  MoveL 1972 to (51.44, -54.38, -208.01) mm, rotated rx -9.61 ry -16.54 rz 125.97 deg; joints [-13.21, -58.037, 110.38, 194.099, 36.852, -114.104, -235]
  MoveL 1973 to (50.7, -54.44, -208.96) mm, rotated rx -9.61 ry -16.54 rz 125.97 deg; joints [-13.251, -58.035, 110.423, 194.018, 36.888, -114.045, -235]
  MoveL 1974 to (50.05, -54.2, -209.74) mm, rotated rx -9.61 ry -16.54 rz 125.97 deg; joints [-13.287, -58.053, 110.472, 193.952, 36.914, -113.997, -235]
  MoveL 1975 to (49.76, -53.97, -210.06) mm, rotated rx -9.61 ry -16.54 rz 125.97 deg; joints [-13.302, -58.07, 110.5, 193.925, 36.922, -113.978, -235]
  MoveL 1976 to (49.49, -53.67, -210.35) mm, rotated rx -9.61 ry -16.54 rz 125.97 deg; joints [-13.316, -58.091, 110.529, 193.901, 36.928, -113.961, -235]
  MoveL 1977 to (49.02, -52.84, -210.78) mm, rotated rx -9.61 ry -16.54 rz 125.97 deg; joints [-13.338, -58.15, 110.594, 193.863, 36.931, -113.936, -235]
  MoveL 1978 to (48.65, -51.71, -211.04) mm, rotated rx -9.61 ry -16.54 rz 125.97 deg; joints [-13.354, -58.228, 110.666, 193.839, 36.922, -113.923, -235]
  MoveL 1979 to (48.37, -50.29, -211.12) mm, rotated rx -9.61 ry -16.54 rz 125.97 deg; joints [-13.364, -58.326, 110.745, 193.83, 36.902, -113.921, -235]
  MoveL 1980 to (48.3, -49.77, -211.12) mm, rotated rx -9.61 ry -16.54 rz 125.97 deg; joints [-13.366, -58.362, 110.773, 193.829, 36.894, -113.922, -235]
  MoveL 1981 to (48.25, -49.32, -211.1) mm, rotated rx -9.61 ry -16.54 rz 125.97 deg; joints [-13.367, -58.393, 110.795, 193.831, 36.885, -113.925, -235]
  MoveL 1982 to (48.22, -48.89, -211.05) mm, rotated rx -9.61 ry -16.54 rz 125.97 deg; joints [-13.367, -58.422, 110.816, 193.834, 36.877, -113.928, -235]
  MoveL 1983 to (48.2, -48.47, -210.99) mm, rotated rx -9.61 ry -16.54 rz 125.97 deg; joints [-13.366, -58.451, 110.835, 193.838, 36.868, -113.933, -235]
  MoveL 1984 to (48.17, -48.02, -210.95) mm, rotated rx -9.61 ry -16.54 rz 125.97 deg; joints [-13.366, -58.482, 110.857, 193.841, 36.859, -113.936, -235]
  MoveL 1985 to (48.11, -47.51, -210.94) mm, rotated rx -9.61 ry -16.54 rz 125.97 deg; joints [-13.367, -58.517, 110.883, 193.842, 36.85, -113.939, -235]
  MoveL 1986 to (48.03, -47, -210.94) mm, rotated rx -9.61 ry -16.54 rz 125.97 deg; joints [-13.37, -58.553, 110.91, 193.841, 36.841, -113.94, -235]
  MoveL 1987 to (47.96, -46.5, -210.93) mm, rotated rx -9.61 ry -16.54 rz 125.97 deg; joints [-13.371, -58.587, 110.936, 193.841, 36.833, -113.941, -235]
  MoveL 1988 to (47.9, -46.03, -210.91) mm, rotated rx -9.61 ry -16.54 rz 125.97 deg; joints [-13.372, -58.619, 110.96, 193.842, 36.825, -113.944, -235]
  MoveL 1989 to (47.87, -45.61, -210.85) mm, rotated rx -9.61 ry -16.54 rz 125.97 deg; joints [-13.372, -58.649, 110.981, 193.845, 36.817, -113.948, -235]
  MoveL 1990 to (47.84, -45.19, -210.79) mm, rotated rx -9.61 ry -16.54 rz 125.97 deg; joints [-13.371, -58.678, 111.001, 193.849, 36.808, -113.952, -235]
  MoveL 1991 to (47.81, -44.72, -210.74) mm, rotated rx -9.61 ry -16.54 rz 125.97 deg; joints [-13.371, -58.71, 111.024, 193.853, 36.799, -113.956, -235]
  MoveL 1992 to (47.74, -44.11, -210.7) mm, rotated rx -9.61 ry -16.54 rz 125.97 deg; joints [-13.372, -58.752, 111.054, 193.855, 36.787, -113.96, -235]
  MoveL 1993 to (47.66, -43.33, -210.68) mm, rotated rx -9.61 ry -16.54 rz 125.97 deg; joints [-13.374, -58.806, 111.093, 193.857, 36.773, -113.964, -235]
  MoveL 1994 to (47.43, -41.77, -210.68) mm, rotated rx -9.61 ry -16.54 rz 125.97 deg; joints [-13.38, -58.913, 111.174, 193.855, 36.746, -113.968, -235]
  MoveL 1995 to (47.32, -40.94, -210.65) mm, rotated rx -9.61 ry -16.54 rz 125.97 deg; joints [-13.383, -58.97, 111.217, 193.856, 36.732, -113.971, -235]
  MoveL 1996 to (47.24, -40.32, -210.64) mm, rotated rx -9.61 ry -16.54 rz 125.97 deg; joints [-13.385, -59.013, 111.248, 193.856, 36.72, -113.974, -235]
  MoveL 1997 to (47.22, -39.83, -210.63) mm, rotated rx -9.61 ry -16.54 rz 125.97 deg; joints [-13.386, -59.046, 111.27, 193.858, 36.709, -113.977, -235]
  MoveL 1998 to (47.24, -39.42, -210.61) mm, rotated rx -9.61 ry -16.54 rz 125.97 deg; joints [-13.387, -59.074, 111.286, 193.861, 36.697, -113.981, -235]
  MoveL 1999 to (47.29, -39.22, -210.5) mm, rotated rx -9.61 ry -16.54 rz 125.97 deg; joints [-13.383, -59.088, 111.291, 193.87, 36.69, -113.989, -235]
  MoveL 2000 to (47.33, -39.28, -210.28) mm, rotated rx -9.61 ry -16.54 rz 125.97 deg; joints [-13.373, -59.085, 111.288, 193.884, 36.692, -113.998, -235]
  MoveL 2001 to (47.35, -39.61, -209.93) mm, rotated rx -9.61 ry -16.54 rz 125.97 deg; joints [-13.358, -59.064, 111.278, 193.905, 36.704, -114.009, -235]
  MoveL 2002 to (48.05, -39.27, -209.23) mm, rotated rx -9.61 ry -16.54 rz 125.97 deg; joints [-13.327, -59.084, 111.248, 193.971, 36.66, -114.06, -235]
  MoveL 2003 to (48.95, -37.47, -209.08) mm, rotated rx -9.61 ry -16.54 rz 125.97 deg; joints [-13.323, -59.194, 111.253, 194.012, 36.558, -114.107, -235]
  MoveL 2004 to (49.84, -35.77, -208.8) mm, rotated rx -9.61 ry -16.54 rz 125.97 deg; joints [-13.312, -59.3, 111.257, 194.062, 36.461, -114.159, -235]
  MoveL 2005 to (50.72, -34.05, -208.52) mm, rotated rx -9.61 ry -16.54 rz 125.97 deg; joints [-13.303, -59.406, 111.262, 194.111, 36.365, -114.21, -235]
  MoveL 2006 to (51.59, -32.32, -208.25) mm, rotated rx -9.61 ry -16.54 rz 125.97 deg; joints [-13.293, -59.513, 111.267, 194.16, 36.268, -114.261, -235]
  MoveL 2007 to (52.5, -30.51, -208.04) mm, rotated rx -9.61 ry -16.54 rz 125.97 deg; joints [-13.286, -59.624, 111.272, 194.207, 36.166, -114.313, -235]
  MoveL 2008 to (53.5, -28.64, -207.89) mm, rotated rx -9.61 ry -16.54 rz 125.97 deg; joints [-13.281, -59.737, 111.271, 194.253, 36.056, -114.366, -235]
  MoveL 2009 to (54.8, -26.46, -207.79) mm, rotated rx -9.61 ry -16.54 rz 125.97 deg; joints [-13.277, -59.867, 111.258, 194.307, 35.918, -114.429, -235]
  MoveL 2010 to (55.75, -24.16, -207.71) mm, rotated rx -9.61 ry -16.54 rz 125.97 deg; joints [-13.277, -60.009, 111.276, 194.35, 35.798, -114.482, -235]
  MoveL 2011 to (56.56, -22.21, -207.6) mm, rotated rx -9.61 ry -16.54 rz 125.97 deg; joints [-13.275, -60.129, 111.291, 194.39, 35.696, -114.529, -235]
  MoveL 2012 to (57.33, -20.48, -207.42) mm, rotated rx -9.61 ry -16.54 rz 125.97 deg; joints [-13.27, -60.236, 111.301, 194.432, 35.603, -114.576, -235]
  MoveL 2013 to (58.2, -18.64, -207.29) mm, rotated rx -9.61 ry -16.54 rz 125.97 deg; joints [-13.266, -60.348, 111.307, 194.475, 35.501, -114.625, -235]
  MoveL 2014 to (59.09, -16.75, -207.16) mm, rotated rx -9.61 ry -16.54 rz 125.97 deg; joints [-13.263, -60.463, 111.312, 194.519, 35.396, -114.676, -235]
  MoveL 2015 to (60.02, -14.79, -207.09) mm, rotated rx -9.61 ry -16.54 rz 125.97 deg; joints [-13.262, -60.581, 111.316, 194.561, 35.285, -114.726, -235]
  MoveL 2016 to (60.93, -12.86, -206.87) mm, rotated rx -9.61 ry -16.54 rz 125.97 deg; joints [-13.255, -60.699, 111.323, 194.613, 35.178, -114.783, -235]
  MoveL 2017 to (61.84, -10.93, -206.75) mm, rotated rx -9.61 ry -16.54 rz 125.97 deg; joints [-13.252, -60.816, 111.327, 194.658, 35.07, -114.835, -235]
  MoveL 2018 to (62.73, -8.99, -206.53) mm, rotated rx -9.61 ry -16.54 rz 125.97 deg; joints [-13.245, -60.934, 111.334, 194.71, 34.963, -114.892, -235]
  MoveL 2019 to (63.64, -7.05, -206.42) mm, rotated rx -9.61 ry -16.54 rz 125.97 deg; joints [-13.242, -61.051, 111.338, 194.755, 34.855, -114.945, -235]
  MoveL 2020 to (64.52, -5.11, -206.2) mm, rotated rx -9.61 ry -16.54 rz 125.97 deg; joints [-13.235, -61.17, 111.345, 194.807, 34.748, -115.002, -235]
  MoveL 2021 to (65.42, -3.18, -206.09) mm, rotated rx -9.61 ry -16.54 rz 125.97 deg; joints [-13.233, -61.286, 111.349, 194.853, 34.64, -115.055, -235]
  MoveL 2022 to (66.32, -1.24, -205.99) mm, rotated rx -9.61 ry -16.54 rz 125.97 deg; joints [-13.23, -61.403, 111.353, 194.899, 34.531, -115.109, -235]
  MoveL 2023 to (67.07, 0.53, -205.75) mm, rotated rx -9.61 ry -16.54 rz 125.97 deg; joints [-13.223, -61.511, 111.363, 194.948, 34.438, -115.162, -235]
  MoveL 2024 to (67.75, 2.22, -205.45) mm, rotated rx -9.61 ry -16.54 rz 125.97 deg; joints [-13.213, -61.616, 111.377, 194.999, 34.351, -115.214, -235]
  MoveL 2025 to (68.37, 3.91, -205.06) mm, rotated rx -9.61 ry -16.54 rz 125.97 deg; joints [-13.2, -61.721, 111.395, 195.055, 34.269, -115.269, -235]
  MoveL 2026 to (67.52, 2.77, -204.14) mm, rotated rx -9.61 ry -16.54 rz 125.97 deg; joints [-13.163, -61.666, 111.432, 195.082, 34.365, -115.268, -235]
  MoveL 2027 to (67.69, 3.1, -204.08) mm, rotated rx -9.61 ry -16.54 rz 125.97 deg; joints [-13.16, -61.685, 111.432, 195.093, 34.346, -115.279, -235]
  MoveL 2028 to (67.88, 3.42, -204.03) mm, rotated rx -9.61 ry -16.54 rz 125.97 deg; joints [-13.158, -61.704, 111.429, 195.105, 34.326, -115.291, -235]
  MoveL 2029 to (68.16, 3.72, -203.99) mm, rotated rx -9.61 ry -16.54 rz 125.97 deg; joints [-13.156, -61.72, 111.419, 195.118, 34.301, -115.306, -235]
  MoveL 2030 to (68.5, 4.02, -203.97) mm, rotated rx -9.61 ry -16.54 rz 125.97 deg; joints [-13.155, -61.735, 111.403, 195.132, 34.272, -115.322, -235]
  MoveL 2031 to (68.92, 4.3, -203.96) mm, rotated rx -9.61 ry -16.54 rz 125.97 deg; joints [-13.153, -61.747, 111.381, 195.148, 34.238, -115.339, -235]
  MoveL 2032 to (69.36, 4.57, -203.96) mm, rotated rx -9.61 ry -16.54 rz 125.97 deg; joints [-13.152, -61.758, 111.357, 195.164, 34.204, -115.358, -235]
  MoveL 2033 to (70.26, 5.11, -203.95) mm, rotated rx -9.61 ry -16.54 rz 125.97 deg; joints [-13.149, -61.78, 111.305, 195.198, 34.134, -115.395, -235]
  MoveL 2034 to (70.67, 5.37, -203.94) mm, rotated rx -9.61 ry -16.54 rz 125.97 deg; joints [-13.147, -61.791, 111.283, 195.214, 34.102, -115.413, -235]
  MoveL 2035 to (71.06, 5.64, -203.89) mm, rotated rx -9.61 ry -16.54 rz 125.97 deg; joints [-13.144, -61.804, 111.263, 195.232, 34.072, -115.431, -235]
  MoveL 2036 to (71.48, 5.95, -203.81) mm, rotated rx -9.61 ry -16.54 rz 125.97 deg; joints [-13.139, -61.818, 111.242, 195.253, 34.038, -115.453, -235]
  MoveL 2037 to (71.96, 6.28, -203.75) mm, rotated rx -9.61 ry -16.54 rz 125.97 deg; joints [-13.136, -61.833, 111.217, 195.275, 34, -115.476, -235]
  MoveL 2038 to (72.44, 6.59, -203.71) mm, rotated rx -9.61 ry -16.54 rz 125.97 deg; joints [-13.133, -61.847, 111.191, 195.295, 33.963, -115.498, -235]
  MoveL 2039 to (72.9, 6.88, -203.7) mm, rotated rx -9.61 ry -16.54 rz 125.97 deg; joints [-13.131, -61.858, 111.165, 195.313, 33.927, -115.518, -235]
  MoveL 2040 to (73.36, 7.15, -203.7) mm, rotated rx -9.61 ry -16.54 rz 125.97 deg; joints [-13.129, -61.869, 111.139, 195.33, 33.891, -115.537, -235]
  MoveL 2041 to (74.26, 7.69, -203.7) mm, rotated rx -9.61 ry -16.54 rz 125.97 deg; joints [-13.126, -61.89, 111.087, 195.364, 33.821, -115.575, -235]
  MoveL 2042 to (75.13, 8.24, -203.67) mm, rotated rx -9.61 ry -16.54 rz 125.97 deg; joints [-13.123, -61.914, 111.039, 195.398, 33.753, -115.613, -235]
  MoveL 2043 to (77.38, 9.58, -203.67) mm, rotated rx -9.61 ry -16.54 rz 125.97 deg; joints [-13.116, -61.966, 110.91, 195.483, 33.579, -115.709, -235]
  MoveL 2044 to (78.65, 10.26, -203.76) mm, rotated rx -9.61 ry -16.54 rz 125.97 deg; joints [-13.115, -61.99, 110.832, 195.525, 33.482, -115.758, -235]
  MoveL 2045 to (79.76, 10.68, -204.02) mm, rotated rx -9.61 ry -16.54 rz 125.97 deg; joints [-13.121, -61.997, 110.756, 195.548, 33.4, -115.792, -235]
  MoveL 2046 to (80.68, 10.84, -204.46) mm, rotated rx -9.61 ry -16.54 rz 125.97 deg; joints [-13.135, -61.989, 110.682, 195.552, 33.334, -115.808, -235]
  MoveL 2047 to (81.08, 10.82, -204.75) mm, rotated rx -9.61 ry -16.54 rz 125.97 deg; joints [-13.144, -61.979, 110.646, 195.546, 33.307, -115.81, -235]
  MoveL 2048 to (81.44, 10.74, -205.08) mm, rotated rx -9.61 ry -16.54 rz 125.97 deg; joints [-13.155, -61.966, 110.611, 195.536, 33.284, -115.808, -235]
  MoveL 2049 to (82.01, 10.37, -205.86) mm, rotated rx -9.61 ry -16.54 rz 125.97 deg; joints [-13.183, -61.926, 110.541, 195.5, 33.251, -115.79, -235]
  MoveL 2050 to (82.42, 9.75, -206.83) mm, rotated rx -9.61 ry -16.54 rz 125.97 deg; joints [-13.218, -61.871, 110.474, 195.445, 33.233, -115.756, -235]
  MoveL 2051 to (82.7, 7.72, -209.29) mm, rotated rx -9.61 ry -16.54 rz 125.97 deg; joints [-13.309, -61.714, 110.345, 195.277, 33.244, -115.636, -235]
  MoveL 2052 to (82.27, 5.33, -211.74) mm, rotated rx -9.61 ry -16.54 rz 125.97 deg; joints [-13.402, -61.544, 110.258, 195.084, 33.308, -115.489, -235]
  MoveL 2053 to (81.14, 3.26, -213.5) mm, rotated rx -9.61 ry -16.54 rz 125.97 deg; joints [-13.471, -61.412, 110.248, 194.917, 33.414, -115.351, -235]
  MoveL 2054 to (80.3, 2.35, -214.11) mm, rotated rx -9.61 ry -16.54 rz 125.97 deg; joints [-13.497, -61.36, 110.272, 194.843, 33.483, -115.285, -235]
  MoveL 2055 to (79.29, 1.51, -214.55) mm, rotated rx -9.61 ry -16.54 rz 125.97 deg; joints [-13.517, -61.318, 110.315, 194.775, 33.562, -115.223, -235]
  MoveL 2056 to (76.74, 0.08, -214.9) mm, rotated rx -9.61 ry -16.54 rz 125.97 deg; joints [-13.54, -61.261, 110.46, 194.659, 33.753, -115.104, -235]
  MoveL 2057 to (74.33, -0.97, -214.9) mm, rotated rx -9.61 ry -16.54 rz 125.97 deg; joints [-13.549, -61.229, 110.611, 194.575, 33.929, -115.011, -235]
  MoveL 2058 to (73.84, -1.17, -214.89) mm, rotated rx -9.61 ry -16.54 rz 125.97 deg; joints [-13.551, -61.223, 110.642, 194.559, 33.965, -114.993, -235]
  MoveL 2059 to (73.34, -1.37, -214.85) mm, rotated rx -9.61 ry -16.54 rz 125.97 deg; joints [-13.552, -61.218, 110.675, 194.543, 34.001, -114.975, -235]
  MoveL 2060 to (72.88, -1.57, -214.85) mm, rotated rx -9.61 ry -16.54 rz 125.97 deg; joints [-13.553, -61.212, 110.704, 194.528, 34.035, -114.958, -235]
  MoveL 2061 to (72.48, -1.75, -214.86) mm, rotated rx -9.61 ry -16.54 rz 125.97 deg; joints [-13.555, -61.206, 110.729, 194.513, 34.064, -114.941, -235]
  MoveL 2062 to (72.03, -1.96, -214.89) mm, rotated rx -9.61 ry -16.54 rz 125.97 deg; joints [-13.558, -61.199, 110.755, 194.496, 34.097, -114.923, -235]
  MoveL 2063 to (71.52, -2.24, -214.96) mm, rotated rx -9.61 ry -16.54 rz 125.97 deg; joints [-13.562, -61.188, 110.785, 194.473, 34.135, -114.9, -235]
  MoveL 2064 to (71.02, -2.51, -215.04) mm, rotated rx -9.61 ry -16.54 rz 125.97 deg; joints [-13.567, -61.177, 110.813, 194.45, 34.172, -114.877, -235]
  MoveL 2065 to (70.51, -2.77, -215.09) mm, rotated rx -9.61 ry -16.54 rz 125.97 deg; joints [-13.571, -61.167, 110.843, 194.429, 34.21, -114.855, -235]
  MoveL 2066 to (70.03, -3, -215.11) mm, rotated rx -9.61 ry -16.54 rz 125.97 deg; joints [-13.574, -61.159, 110.872, 194.411, 34.245, -114.836, -235]
  MoveL 2067 to (69.56, -3.21, -215.12) mm, rotated rx -9.61 ry -16.54 rz 125.97 deg; joints [-13.576, -61.152, 110.901, 194.395, 34.28, -114.818, -235]
  MoveL 2068 to (69.08, -3.42, -215.12) mm, rotated rx -9.61 ry -16.54 rz 125.97 deg; joints [-13.578, -61.145, 110.931, 194.378, 34.315, -114.799, -235]
  MoveL 2069 to (68.57, -3.67, -215.15) mm, rotated rx -9.61 ry -16.54 rz 125.97 deg; joints [-13.581, -61.136, 110.961, 194.358, 34.352, -114.779, -235]
  MoveL 2070 to (68.08, -3.93, -215.2) mm, rotated rx -9.61 ry -16.54 rz 125.97 deg; joints [-13.585, -61.126, 110.989, 194.338, 34.389, -114.758, -235]
  MoveL 2071 to (67.6, -4.21, -215.27) mm, rotated rx -9.61 ry -16.54 rz 125.97 deg; joints [-13.589, -61.114, 111.015, 194.317, 34.425, -114.736, -235]
  MoveL 2072 to (67.19, -4.51, -215.33) mm, rotated rx -9.61 ry -16.54 rz 125.97 deg; joints [-13.593, -61.1, 111.035, 194.299, 34.458, -114.717, -235]
  MoveL 2073 to (66.84, -4.81, -215.36) mm, rotated rx -9.61 ry -16.54 rz 125.97 deg; joints [-13.595, -61.084, 111.05, 194.284, 34.487, -114.701, -235]
  MoveL 2074 to (66.59, -5.13, -215.37) mm, rotated rx -9.61 ry -16.54 rz 125.97 deg; joints [-13.596, -61.067, 111.059, 194.274, 34.512, -114.69, -235]
  MoveL 2075 to (66.37, -5.45, -215.37) mm, rotated rx -9.61 ry -16.54 rz 125.97 deg; joints [-13.596, -61.049, 111.064, 194.266, 34.534, -114.679, -235]
  MoveL 2076 to (67.23, -4.49, -216.25) mm, rotated rx -9.61 ry -16.54 rz 125.97 deg; joints [-13.63, -61.093, 111.02, 194.24, 34.443, -114.68, -235]
  MoveL 2077 to (66.47, -5.9, -216.53) mm, rotated rx -9.61 ry -16.54 rz 125.97 deg; joints [-13.64, -61.009, 111.022, 194.191, 34.526, -114.631, -235]
  MoveL 2078 to (65.57, -7.46, -216.73) mm, rotated rx -9.61 ry -16.54 rz 125.97 deg; joints [-13.647, -60.917, 111.032, 194.143, 34.624, -114.579, -235]
  MoveL 2079 to (64.5, -9.21, -216.86) mm, rotated rx -9.61 ry -16.54 rz 125.97 deg; joints [-13.652, -60.815, 111.047, 194.094, 34.737, -114.523, -235]
  MoveL 2080 to (63.3, -11.12, -216.95) mm, rotated rx -9.61 ry -16.54 rz 125.97 deg; joints [-13.656, -60.704, 111.067, 194.043, 34.862, -114.464, -235]
  MoveL 2081 to (62.18, -12.93, -217.1) mm, rotated rx -9.61 ry -16.54 rz 125.97 deg; joints [-13.661, -60.598, 111.083, 193.991, 34.98, -114.407, -235]
  MoveL 2082 to (61.06, -14.76, -217.31) mm, rotated rx -9.61 ry -16.54 rz 125.97 deg; joints [-13.669, -60.491, 111.097, 193.936, 35.097, -114.347, -235]
  MoveL 2083 to (59.99, -16.48, -217.43) mm, rotated rx -9.61 ry -16.54 rz 125.97 deg; joints [-13.674, -60.39, 111.112, 193.889, 35.209, -114.294, -235]
  MoveL 2084 to (59.04, -18.06, -217.69) mm, rotated rx -9.61 ry -16.54 rz 125.97 deg; joints [-13.684, -60.296, 111.122, 193.837, 35.308, -114.24, -235]
  MoveL 2085 to (57.95, -19.82, -217.91) mm, rotated rx -9.61 ry -16.54 rz 125.97 deg; joints [-13.693, -60.192, 111.136, 193.783, 35.421, -114.182, -235]
  MoveL 2086 to (56.84, -21.58, -218.05) mm, rotated rx -9.61 ry -16.54 rz 125.97 deg; joints [-13.698, -60.088, 111.151, 193.735, 35.536, -114.128, -235]
  MoveL 2087 to (55.69, -23.38, -218.15) mm, rotated rx -9.61 ry -16.54 rz 125.97 deg; joints [-13.702, -59.982, 111.168, 193.688, 35.654, -114.074, -235]
  MoveL 2088 to (54.57, -25.18, -218.38) mm, rotated rx -9.61 ry -16.54 rz 125.97 deg; joints [-13.711, -59.876, 111.182, 193.634, 35.77, -114.016, -235]
  MoveL 2089 to (53.4, -26.98, -218.64) mm, rotated rx -9.61 ry -16.54 rz 125.97 deg; joints [-13.721, -59.769, 111.197, 193.577, 35.888, -113.956, -235]
  MoveL 2090 to (52.25, -28.77, -218.73) mm, rotated rx -9.61 ry -16.54 rz 125.97 deg; joints [-13.725, -59.663, 111.214, 193.532, 36.006, -113.903, -235]
  MoveL 2091 to (51.08, -30.6, -218.77) mm, rotated rx -9.61 ry -16.54 rz 125.97 deg; joints [-13.726, -59.555, 111.231, 193.489, 36.127, -113.852, -235]
  MoveL 2092 to (49.94, -32.38, -218.88) mm, rotated rx -9.61 ry -16.54 rz 125.97 deg; joints [-13.73, -59.45, 111.247, 193.444, 36.245, -113.8, -235]
  MoveL 2093 to (48.78, -34.16, -219.08) mm, rotated rx -9.61 ry -16.54 rz 125.97 deg; joints [-13.738, -59.344, 111.263, 193.393, 36.361, -113.744, -235]
  MoveL 2094 to (47.64, -35.89, -219.42) mm, rotated rx -9.61 ry -16.54 rz 125.97 deg; joints [-13.752, -59.24, 111.276, 193.334, 36.474, -113.685, -235]
  MoveL 2095 to (46.43, -37.68, -219.67) mm, rotated rx -9.61 ry -16.54 rz 125.97 deg; joints [-13.762, -59.133, 111.293, 193.279, 36.593, -113.626, -235]
  MoveL 2096 to (45.24, -39.45, -219.88) mm, rotated rx -9.61 ry -16.54 rz 125.97 deg; joints [-13.771, -59.027, 111.31, 193.228, 36.712, -113.571, -235]
  MoveL 2097 to (44.02, -41.25, -220.11) mm, rotated rx -9.61 ry -16.54 rz 125.97 deg; joints [-13.781, -58.919, 111.327, 193.174, 36.832, -113.513, -235]
  MoveL 2098 to (42.83, -43.04, -220.26) mm, rotated rx -9.61 ry -16.54 rz 125.97 deg; joints [-13.786, -58.812, 111.343, 193.127, 36.952, -113.461, -235]
  MoveL 2099 to (41.68, -44.82, -220.28) mm, rotated rx -9.61 ry -16.54 rz 125.97 deg; joints [-13.787, -58.705, 111.358, 193.09, 37.069, -113.415, -235]
  MoveL 2100 to (41.09, -45.06, -220.94) mm, rotated rx -9.61 ry -16.54 rz 125.97 deg; joints [-13.816, -58.691, 111.384, 193.032, 37.104, -113.371, -235]
  MoveL 2101 to (41.2, -44.74, -221.27) mm, rotated rx -9.61 ry -16.54 rz 125.97 deg; joints [-13.83, -58.709, 111.384, 193.015, 37.086, -113.364, -235]
  MoveL 2102 to (41.2, -44.7, -221.48) mm, rotated rx -9.61 ry -16.54 rz 125.97 deg; joints [-13.839, -58.71, 111.383, 193.003, 37.082, -113.357, -235]
  MoveL 2103 to (41.13, -44.9, -221.58) mm, rotated rx -9.61 ry -16.54 rz 125.97 deg; joints [-13.842, -58.696, 111.378, 192.994, 37.09, -113.349, -235]
  MoveL 2104 to (41.05, -45.32, -221.6) mm, rotated rx -9.61 ry -16.54 rz 125.97 deg; joints [-13.842, -58.669, 111.367, 192.99, 37.106, -113.344, -235]
  MoveC 2105 to (41.01, -46.33, -221.6) mm, rotated rx -9.61 ry -16.54 rz 125.97 deg; joints [-13.839, -58.601, 111.329, 192.986, 37.135, -113.336, -235] to (41.03, -47.35, -221.6) mm, rotated rx -9.61 ry -16.54 rz 125.97 deg; joints [-13.835, -58.533, 111.285, 192.985, 37.16, -113.331, -235]
  MoveL 2106 to (41.03, -47.35, -221.61) mm, rotated rx -9.61 ry -16.54 rz 125.97 deg; joints [-13.835, -58.533, 111.285, 192.985, 37.16, -113.33, -235]
  MoveL 2107 to (41.03, -47.9, -221.63) mm, rotated rx -9.61 ry -16.54 rz 125.97 deg; joints [-13.834, -58.496, 111.262, 192.982, 37.174, -113.326, -235]
  MoveL 2108 to (41.01, -48.43, -221.68) mm, rotated rx -9.61 ry -16.54 rz 125.97 deg; joints [-13.834, -58.459, 111.241, 192.978, 37.188, -113.321, -235]
  MoveL 2109 to (40.98, -49.01, -221.75) mm, rotated rx -9.61 ry -16.54 rz 125.97 deg; joints [-13.835, -58.42, 111.218, 192.971, 37.204, -113.314, -235]
  MoveL 2110 to (40.97, -49.61, -221.79) mm, rotated rx -9.61 ry -16.54 rz 125.97 deg; joints [-13.834, -58.38, 111.194, 192.967, 37.22, -113.308, -235]
  MoveL 2111 to (40.97, -50.82, -221.81) mm, rotated rx -9.61 ry -16.54 rz 125.97 deg; joints [-13.831, -58.298, 111.142, 192.964, 37.25, -113.3, -235]
  MoveL 2112 to (40.96, -51.38, -221.84) mm, rotated rx -9.61 ry -16.54 rz 125.97 deg; joints [-13.83, -58.261, 111.12, 192.961, 37.265, -113.295, -235]
  MoveL 2113 to (40.93, -51.85, -221.92) mm, rotated rx -9.61 ry -16.54 rz 125.97 deg; joints [-13.832, -58.229, 111.102, 192.954, 37.278, -113.289, -235]
  MoveL 2114 to (40.88, -52.29, -222.01) mm, rotated rx -9.61 ry -16.54 rz 125.97 deg; joints [-13.834, -58.199, 111.086, 192.947, 37.291, -113.282, -235]
  MoveL 2115 to (40.85, -52.71, -222.07) mm, rotated rx -9.61 ry -16.54 rz 125.97 deg; joints [-13.835, -58.171, 111.07, 192.941, 37.303, -113.276, -235]
  MoveL 2116 to (40.84, -53.16, -222.1) mm, rotated rx -9.61 ry -16.54 rz 125.97 deg; joints [-13.835, -58.14, 111.051, 192.938, 37.315, -113.272, -235]
  MoveL 2117 to (40.9, -55.78, -222.1) mm, rotated rx -9.61 ry -16.54 rz 125.97 deg; joints [-13.825, -57.963, 110.937, 192.935, 37.377, -113.258, -235]
  MoveL 2118 to (40.69, -58.68, -222.45) mm, rotated rx -9.61 ry -16.54 rz 125.97 deg; joints [-13.83, -57.768, 110.826, 192.903, 37.459, -113.222, -235]
  MoveL 2119 to (40.38, -59.92, -222.88) mm, rotated rx -9.61 ry -16.54 rz 125.97 deg; joints [-13.844, -57.685, 110.791, 192.866, 37.504, -113.191, -235]
  MoveL 2120 to (39.93, -61.03, -223.48) mm, rotated rx -9.61 ry -16.54 rz 125.97 deg; joints [-13.867, -57.611, 110.77, 192.816, 37.553, -113.15, -235]
  MoveL 2121 to (39.34, -62, -224.26) mm, rotated rx -9.61 ry -16.54 rz 125.97 deg; joints [-13.898, -57.546, 110.763, 192.751, 37.605, -113.099, -235]
  MoveL 2122 to (38.61, -62.84, -225.21) mm, rotated rx -9.61 ry -16.54 rz 125.97 deg; joints [-13.936, -57.491, 110.77, 192.673, 37.66, -113.04, -235]
  MoveL 2123 to (36.73, -64.09, -227.62) mm, rotated rx -9.61 ry -16.54 rz 125.97 deg; joints [-14.039, -57.408, 110.824, 192.475, 37.78, -112.894, -235]
  MoveL 2124 to (34.88, -64.56, -230.04) mm, rotated rx -9.61 ry -16.54 rz 125.97 deg; joints [-14.144, -57.378, 110.909, 192.28, 37.88, -112.754, -235]
  MoveL 2125 to (34.19, -64.4, -230.99) mm, rotated rx -9.61 ry -16.54 rz 125.97 deg; joints [-14.186, -57.388, 110.954, 192.205, 37.908, -112.702, -235]
  MoveL 2126 to (33.65, -63.99, -231.76) mm, rotated rx -9.61 ry -16.54 rz 125.97 deg; joints [-14.222, -57.416, 111.001, 192.144, 37.923, -112.661, -235]
  MoveL 2127 to (33.44, -63.68, -232.08) mm, rotated rx -9.61 ry -16.54 rz 125.97 deg; joints [-14.237, -57.436, 111.026, 192.119, 37.925, -112.645, -235]
  MoveL 2128 to (33.27, -63.31, -232.36) mm, rotated rx -9.61 ry -16.54 rz 125.97 deg; joints [-14.251, -57.461, 111.05, 192.098, 37.923, -112.632, -235]
  MoveL 2129 to (33.04, -62.38, -232.8) mm, rotated rx -9.61 ry -16.54 rz 125.97 deg; joints [-14.273, -57.523, 111.101, 192.067, 37.909, -112.615, -235]
  MoveL 2130 to (32.97, -61.19, -233.05) mm, rotated rx -9.61 ry -16.54 rz 125.97 deg; joints [-14.289, -57.602, 111.153, 192.05, 37.881, -112.61, -235]
  MoveL 2131 to (33.05, -59.74, -233.14) mm, rotated rx -9.61 ry -16.54 rz 125.97 deg; joints [-14.297, -57.698, 111.207, 192.048, 37.839, -112.616, -235]
  MoveL 2132 to (33.1, -59.22, -233.14) mm, rotated rx -9.61 ry -16.54 rz 125.97 deg; joints [-14.299, -57.732, 111.225, 192.05, 37.823, -112.62, -235]
  MoveL 2133 to (33.16, -58.77, -233.11) mm, rotated rx -9.61 ry -16.54 rz 125.97 deg; joints [-14.299, -57.762, 111.24, 192.054, 37.808, -112.625, -235]
  MoveL 2134 to (33.24, -58.36, -233.05) mm, rotated rx -9.61 ry -16.54 rz 125.97 deg; joints [-14.298, -57.789, 111.252, 192.06, 37.793, -112.631, -235]
  MoveL 2135 to (33.32, -57.96, -232.98) mm, rotated rx -9.61 ry -16.54 rz 125.97 deg; joints [-14.296, -57.816, 111.264, 192.067, 37.779, -112.638, -235]
  MoveL 2136 to (33.4, -57.53, -232.94) mm, rotated rx -9.61 ry -16.54 rz 125.97 deg; joints [-14.295, -57.845, 111.277, 192.072, 37.764, -112.644, -235]
  MoveL 2137 to (33.46, -57.02, -232.92) mm, rotated rx -9.61 ry -16.54 rz 125.97 deg; joints [-14.296, -57.878, 111.294, 192.075, 37.748, -112.649, -235]
  MoveL 2138 to (34.03, -51.32, -232.91) mm, rotated rx -9.61 ry -16.54 rz 125.97 deg; joints [-14.314, -58.256, 111.49, 192.096, 37.567, -112.694, -235]
  MoveL 2139 to (34.12, -50.56, -232.89) mm, rotated rx -9.61 ry -16.54 rz 125.97 deg; joints [-14.316, -58.307, 111.515, 192.1, 37.542, -112.701, -235]
  MoveL 2140 to (34.23, -49.91, -232.89) mm, rotated rx -9.61 ry -16.54 rz 125.97 deg; joints [-14.318, -58.349, 111.534, 192.104, 37.519, -112.708, -235]
  MoveL 2141 to (34.4, -49.37, -232.87) mm, rotated rx -9.61 ry -16.54 rz 125.97 deg; joints [-14.318, -58.384, 111.543, 192.111, 37.493, -112.716, -235]
  MoveL 2142 to (34.64, -48.88, -232.83) mm, rotated rx -9.61 ry -16.54 rz 125.97 deg; joints [-14.317, -58.415, 111.546, 192.12, 37.467, -112.727, -235]
  MoveL 2143 to (34.83, -48.61, -232.67) mm, rotated rx -9.61 ry -16.54 rz 125.97 deg; joints [-14.311, -58.432, 111.545, 192.135, 37.449, -112.739, -235]
  MoveL 2144 to (34.85, -48.63, -232.36) mm, rotated rx -9.61 ry -16.54 rz 125.97 deg; joints [-14.298, -58.433, 111.547, 192.155, 37.452, -112.751, -235]
  MoveL 2145 to (34.68, -48.95, -231.88) mm, rotated rx -9.61 ry -16.54 rz 125.97 deg; joints [-14.278, -58.417, 111.554, 192.179, 37.477, -112.762, -235]
  MoveL 2146 to (35.3, -49.04, -230.91) mm, rotated rx -9.61 ry -16.54 rz 125.97 deg; joints [-14.235, -58.412, 111.517, 192.255, 37.452, -112.815, -235]
  MoveL 2147 to (36.53, -47.63, -230.61) mm, rotated rx -9.61 ry -16.54 rz 125.97 deg; joints [-14.221, -58.496, 111.487, 192.309, 37.342, -112.868, -235]
  MoveL 2148 to (37.8, -46.13, -230.4) mm, rotated rx -9.61 ry -16.54 rz 125.97 deg; joints [-14.211, -58.583, 111.455, 192.358, 37.226, -112.92, -235]
  MoveL 2149 to (39.17, -44.5, -230.27) mm, rotated rx -9.61 ry -16.54 rz 125.97 deg; joints [-14.205, -58.678, 111.419, 192.405, 37.1, -112.973, -235]
  MoveL 2150 to (41.88, -41.21, -230.27) mm, rotated rx -9.61 ry -16.54 rz 125.97 deg; joints [-14.202, -58.867, 111.346, 192.485, 36.844, -113.07, -235]
  MoveL 2151 to (43.14, -39.68, -230.18) mm, rotated rx -9.61 ry -16.54 rz 125.97 deg; joints [-14.197, -58.956, 111.313, 192.528, 36.726, -113.119, -235]
  MoveL 2152 to (44.5, -38.04, -230.18) mm, rotated rx -9.61 ry -16.54 rz 125.97 deg; joints [-14.195, -59.05, 111.276, 192.569, 36.598, -113.168, -235]
  MoveL 2153 to (45.95, -36.43, -230.18) mm, rotated rx -9.61 ry -16.54 rz 125.97 deg; joints [-14.193, -59.139, 111.229, 192.613, 36.465, -113.22, -235]
  MoveL 2154 to (47.68, -34.57, -230.01) mm, rotated rx -9.61 ry -16.54 rz 125.97 deg; joints [-14.183, -59.244, 111.173, 192.677, 36.31, -113.29, -235]
  MoveL 2155 to (49, -32.78, -229.77) mm, rotated rx -9.61 ry -16.54 rz 125.97 deg; joints [-14.173, -59.349, 111.147, 192.732, 36.183, -113.349, -235]
  MoveL 2156 to (50.3, -31.04, -229.65) mm, rotated rx -9.61 ry -16.54 rz 125.97 deg; joints [-14.167, -59.45, 111.118, 192.781, 36.057, -113.403, -235]
  MoveL 2157 to (51.66, -29.39, -229.55) mm, rotated rx -9.61 ry -16.54 rz 125.97 deg; joints [-14.161, -59.544, 111.08, 192.83, 35.93, -113.459, -235]
  MoveL 2158 to (53.01, -27.74, -229.33) mm, rotated rx -9.61 ry -16.54 rz 125.97 deg; joints [-14.151, -59.638, 111.044, 192.887, 35.804, -113.519, -235]
  MoveL 2159 to (54.36, -26.09, -229.22) mm, rotated rx -9.61 ry -16.54 rz 125.97 deg; joints [-14.145, -59.731, 111.006, 192.937, 35.677, -113.575, -235]
  MoveL 2160 to (55.71, -24.44, -229.11) mm, rotated rx -9.61 ry -16.54 rz 125.97 deg; joints [-14.139, -59.824, 110.968, 192.988, 35.55, -113.632, -235]
  MoveL 2161 to (57.05, -22.78, -228.9) mm, rotated rx -9.61 ry -16.54 rz 125.97 deg; joints [-14.129, -59.919, 110.932, 193.045, 35.425, -113.693, -235]
  MoveL 2162 to (58.4, -21.12, -228.8) mm, rotated rx -9.61 ry -16.54 rz 125.97 deg; joints [-14.124, -60.012, 110.894, 193.096, 35.298, -113.75, -235]
  MoveL 2163 to (59.75, -19.47, -228.69) mm, rotated rx -9.61 ry -16.54 rz 125.97 deg; joints [-14.118, -60.104, 110.855, 193.148, 35.171, -113.808, -235]
  MoveL 2164 to (61.07, -17.8, -228.48) mm, rotated rx -9.61 ry -16.54 rz 125.97 deg; joints [-14.109, -60.198, 110.819, 193.206, 35.045, -113.87, -235]
  MoveL 2165 to (62.42, -16.14, -228.38) mm, rotated rx -9.61 ry -16.54 rz 125.97 deg; joints [-14.103, -60.291, 110.78, 193.258, 34.918, -113.928, -235]
  MoveL 2166 to (63.52, -14.66, -228.12) mm, rotated rx -9.61 ry -16.54 rz 125.97 deg; joints [-14.092, -60.376, 110.755, 193.313, 34.812, -113.984, -235]
  MoveL 2167 to (64.47, -13.28, -227.76) mm, rotated rx -9.61 ry -16.54 rz 125.97 deg; joints [-14.077, -60.456, 110.738, 193.37, 34.72, -114.04, -235]
  MoveL 2168 to (65.28, -11.99, -227.26) mm, rotated rx -9.61 ry -16.54 rz 125.97 deg; joints [-14.057, -60.535, 110.732, 193.431, 34.641, -114.096, -235]
  MoveL 2169 to (64.38, -12.68, -226.41) mm, rotated rx -9.61 ry -16.54 rz 125.97 deg; joints [-14.026, -60.509, 110.788, 193.456, 34.725, -114.097, -235]
  MoveL 2170 to (64.59, -12.43, -226.38) mm, rotated rx -9.61 ry -16.54 rz 125.97 deg; joints [-14.024, -60.523, 110.782, 193.465, 34.706, -114.107, -235]
  MoveL 2171 to (64.82, -12.2, -226.34) mm, rotated rx -9.61 ry -16.54 rz 125.97 deg; joints [-14.022, -60.535, 110.773, 193.476, 34.686, -114.118, -235]
  MoveL 2172 to (65.14, -12.01, -226.29) mm, rotated rx -9.61 ry -16.54 rz 125.97 deg; joints [-14.019, -60.543, 110.757, 193.49, 34.662, -114.132, -235]
  MoveL 2173 to (65.51, -11.83, -226.25) mm, rotated rx -9.61 ry -16.54 rz 125.97 deg; joints [-14.016, -60.55, 110.734, 193.505, 34.634, -114.147, -235]
  MoveL 2174 to (65.97, -11.67, -226.22) mm, rotated rx -9.61 ry -16.54 rz 125.97 deg; joints [-14.013, -60.555, 110.705, 193.521, 34.602, -114.164, -235]
  MoveL 2175 to (70.48, -10.31, -226.22) mm, rotated rx -9.61 ry -16.54 rz 125.97 deg; joints [-13.993, -60.577, 110.402, 193.667, 34.288, -114.322, -235]
  MoveL 2176 to (70.86, -10.18, -226.2) mm, rotated rx -9.61 ry -16.54 rz 125.97 deg; joints [-13.99, -60.581, 110.378, 193.681, 34.262, -114.336, -235]
  MoveL 2177 to (71.36, -10.03, -226.2) mm, rotated rx -9.61 ry -16.54 rz 125.97 deg; joints [-13.988, -60.583, 110.344, 193.697, 34.227, -114.354, -235]
  MoveL 2178 to (72.34, -9.71, -226.16) mm, rotated rx -9.61 ry -16.54 rz 125.97 deg; joints [-13.982, -60.59, 110.28, 193.732, 34.159, -114.391, -235]
  MoveL 2179 to (74.85, -8.96, -226.16) mm, rotated rx -9.61 ry -16.54 rz 125.97 deg; joints [-13.971, -60.601, 110.11, 193.815, 33.985, -114.48, -235]
  MoveL 2180 to (75.82, -8.61, -226.14) mm, rotated rx -9.61 ry -16.54 rz 125.97 deg; joints [-13.966, -60.61, 110.047, 193.848, 33.916, -114.516, -235]
  MoveL 2181 to (77.2, -8.17, -226.21) mm, rotated rx -9.61 ry -16.54 rz 125.97 deg; joints [-13.962, -60.616, 109.953, 193.89, 33.819, -114.563, -235]
  MoveL 2182 to (78.35, -7.96, -226.46) mm, rotated rx -9.61 ry -16.54 rz 125.97 deg; joints [-13.967, -60.61, 109.866, 193.911, 33.74, -114.593, -235]
  MoveL 2183 to (79.28, -7.97, -226.9) mm, rotated rx -9.61 ry -16.54 rz 125.97 deg; joints [-13.979, -60.591, 109.786, 193.912, 33.678, -114.605, -235]
  MoveL 2184 to (79.66, -8.06, -227.19) mm, rotated rx -9.61 ry -16.54 rz 125.97 deg; joints [-13.988, -60.577, 109.748, 193.905, 33.654, -114.605, -235]
  MoveL 2185 to (79.99, -8.2, -227.53) mm, rotated rx -9.61 ry -16.54 rz 125.97 deg; joints [-14, -60.56, 109.712, 193.893, 33.634, -114.6, -235]
  MoveL 2186 to (80.46, -8.65, -228.34) mm, rotated rx -9.61 ry -16.54 rz 125.97 deg; joints [-14.028, -60.516, 109.645, 193.853, 33.608, -114.578, -235]
  MoveL 2187 to (80.72, -9.33, -229.34) mm, rotated rx -9.61 ry -16.54 rz 125.97 deg; joints [-14.064, -60.459, 109.585, 193.792, 33.599, -114.538, -235]
  MoveL 2188 to (80.55, -11.33, -231.89) mm, rotated rx -9.61 ry -16.54 rz 125.97 deg; joints [-14.159, -60.308, 109.485, 193.611, 33.633, -114.407, -235]
  MoveL 2189 to (79.61, -13.54, -234.46) mm, rotated rx -9.61 ry -16.54 rz 125.97 deg; joints [-14.258, -60.155, 109.436, 193.404, 33.72, -114.249, -235]
  MoveL 2190 to (78.05, -15.28, -236.29) mm, rotated rx -9.61 ry -16.54 rz 125.97 deg; joints [-14.334, -60.049, 109.466, 193.229, 33.84, -114.107, -235]
  MoveL 2191 to (77.03, -15.97, -236.93) mm, rotated rx -9.61 ry -16.54 rz 125.97 deg; joints [-14.362, -60.014, 109.51, 193.153, 33.913, -114.042, -235]
  MoveL 2192 to (75.86, -16.54, -237.39) mm, rotated rx -9.61 ry -16.54 rz 125.97 deg; joints [-14.385, -59.99, 109.574, 193.085, 33.995, -113.981, -235]
  MoveL 2193 to (73.05, -17.32, -237.76) mm, rotated rx -9.61 ry -16.54 rz 125.97 deg; joints [-14.413, -59.978, 109.76, 192.972, 34.185, -113.87, -235]
  MoveL 2194 to (69.95, -17.86, -237.76) mm, rotated rx -9.61 ry -16.54 rz 125.97 deg; joints [-14.429, -59.988, 109.983, 192.875, 34.389, -113.768, -235]
  MoveL 2195 to (68.96, -18.06, -237.77) mm, rotated rx -9.61 ry -16.54 rz 125.97 deg; joints [-14.434, -59.99, 110.053, 192.844, 34.456, -113.734, -235]
  MoveL 2196 to (67.92, -18.24, -237.77) mm, rotated rx -9.61 ry -16.54 rz 125.97 deg; joints [-14.44, -59.993, 110.127, 192.812, 34.524, -113.701, -235]
  MoveL 2197 to (67.43, -18.33, -237.77) mm, rotated rx -9.61 ry -16.54 rz 125.97 deg; joints [-14.443, -59.994, 110.162, 192.796, 34.557, -113.684, -235]
  MoveL 2198 to (66.78, -18.46, -237.8) mm, rotated rx -9.61 ry -16.54 rz 125.97 deg; joints [-14.447, -59.995, 110.208, 192.774, 34.6, -113.662, -235]
  MoveL 2199 to (66.2, -18.59, -237.86) mm, rotated rx -9.61 ry -16.54 rz 125.97 deg; joints [-14.452, -59.994, 110.248, 192.753, 34.639, -113.64, -235]
  MoveL 2200 to (65.71, -18.72, -237.93) mm, rotated rx -9.61 ry -16.54 rz 125.97 deg; joints [-14.457, -59.992, 110.28, 192.733, 34.671, -113.622, -235]
  MoveL 2201 to (65.26, -18.83, -237.99) mm, rotated rx -9.61 ry -16.54 rz 125.97 deg; joints [-14.462, -59.99, 110.31, 192.716, 34.701, -113.605, -235]
  MoveL 2202 to (64.81, -18.93, -238.02) mm, rotated rx -9.61 ry -16.54 rz 125.97 deg; joints [-14.465, -59.99, 110.341, 192.7, 34.732, -113.589, -235]
  MoveL 2203 to (63.26, -19.2, -238.02) mm, rotated rx -9.61 ry -16.54 rz 125.97 deg; joints [-14.473, -59.994, 110.452, 192.653, 34.834, -113.539, -235]
  MoveL 2204 to (62.77, -19.31, -238.03) mm, rotated rx -9.61 ry -16.54 rz 125.97 deg; joints [-14.476, -59.994, 110.486, 192.637, 34.867, -113.522, -235]
  MoveL 2205 to (62.35, -19.42, -238.06) mm, rotated rx -9.61 ry -16.54 rz 125.97 deg; joints [-14.479, -59.992, 110.514, 192.622, 34.896, -113.507, -235]
  MoveL 2206 to (61.98, -19.56, -238.11) mm, rotated rx -9.61 ry -16.54 rz 125.97 deg; joints [-14.483, -59.988, 110.537, 192.608, 34.922, -113.494, -235]
  MoveL 2207 to (61.72, -19.71, -238.17) mm, rotated rx -9.61 ry -16.54 rz 125.97 deg; joints [-14.486, -59.981, 110.549, 192.596, 34.941, -113.482, -235]
  MoveL 2208 to (61.52, -19.89, -238.24) mm, rotated rx -9.61 ry -16.54 rz 125.97 deg; joints [-14.49, -59.971, 110.558, 192.585, 34.958, -113.472, -235]
  MoveL 2209 to (63.02, -19.39, -239.05) mm, rotated rx -9.61 ry -16.54 rz 125.97 deg; joints [-14.515, -59.976, 110.447, 192.579, 34.842, -113.488, -235]
  MoveL 2210 to (61.72, -20.58, -239.45) mm, rotated rx -9.61 ry -16.54 rz 125.97 deg; joints [-14.534, -59.912, 110.497, 192.512, 34.95, -113.424, -235]
  MoveL 2211 to (60.36, -21.87, -239.71) mm, rotated rx -9.61 ry -16.54 rz 125.97 deg; joints [-14.548, -59.843, 110.549, 192.452, 35.066, -113.364, -235]
  MoveL 2212 to (58.92, -23.27, -239.9) mm, rotated rx -9.61 ry -16.54 rz 125.97 deg; joints [-14.558, -59.769, 110.603, 192.396, 35.191, -113.305, -235]
  MoveL 2213 to (57.4, -24.77, -240.09) mm, rotated rx -9.61 ry -16.54 rz 125.97 deg; joints [-14.569, -59.688, 110.659, 192.336, 35.323, -113.243, -235]
  MoveL 2214 to (55.87, -26.25, -240.18) mm, rotated rx -9.61 ry -16.54 rz 125.97 deg; joints [-14.576, -59.609, 110.718, 192.283, 35.457, -113.184, -235]
  MoveL 2215 to (54.34, -27.74, -240.28) mm, rotated rx -9.61 ry -16.54 rz 125.97 deg; joints [-14.583, -59.529, 110.777, 192.231, 35.591, -113.126, -235]
  MoveL 2216 to (52.81, -29.23, -240.48) mm, rotated rx -9.61 ry -16.54 rz 125.97 deg; joints [-14.594, -59.448, 110.833, 192.172, 35.723, -113.065, -235]
  MoveL 2217 to (51.28, -30.71, -240.58) mm, rotated rx -9.61 ry -16.54 rz 125.97 deg; joints [-14.601, -59.369, 110.891, 192.12, 35.858, -113.008, -235]
  MoveL 2218 to (49.74, -32.19, -240.68) mm, rotated rx -9.61 ry -16.54 rz 125.97 deg; joints [-14.609, -59.289, 110.949, 192.068, 35.991, -112.951, -235]
  MoveL 2219 to (48.2, -33.67, -240.88) mm, rotated rx -9.61 ry -16.54 rz 125.97 deg; joints [-14.62, -59.207, 111.005, 192.011, 36.124, -112.891, -235]
  MoveL 2220 to (45.12, -36.63, -241.08) mm, rotated rx -9.61 ry -16.54 rz 125.97 deg; joints [-14.635, -59.046, 111.12, 191.909, 36.392, -112.779, -235]
  MoveL 2221 to (43.83, -37.86, -241.29) mm, rotated rx -9.61 ry -16.54 rz 125.97 deg; joints [-14.646, -58.978, 111.167, 191.859, 36.504, -112.728, -235]
  MoveL 2222 to (42.44, -39.25, -241.36) mm, rotated rx -9.61 ry -16.54 rz 125.97 deg; joints [-14.652, -58.901, 111.216, 191.815, 36.626, -112.679, -235]
  MoveL 2223 to (41.02, -40.74, -241.37) mm, rotated rx -9.61 ry -16.54 rz 125.97 deg; joints [-14.655, -58.818, 111.264, 191.775, 36.754, -112.631, -235]
  MoveL 2224 to (39.08, -42.58, -241.48) mm, rotated rx -9.61 ry -16.54 rz 125.97 deg; joints [-14.663, -58.717, 111.335, 191.714, 36.922, -112.563, -235]
  MoveL 2225 to (37.13, -44.27, -241.58) mm, rotated rx -9.61 ry -16.54 rz 125.97 deg; joints [-14.672, -58.625, 111.413, 191.655, 37.087, -112.498, -235]
  MoveL 2226 to (35.51, -45.76, -241.67) mm, rotated rx -9.61 ry -16.54 rz 125.97 deg; joints [-14.68, -58.542, 111.475, 191.604, 37.227, -112.442, -235]
  MoveL 2227 to (34.01, -47.16, -241.84) mm, rotated rx -9.61 ry -16.54 rz 125.97 deg; joints [-14.69, -58.464, 111.528, 191.553, 37.355, -112.389, -235]
  MoveL 2228 to (32.61, -48.45, -242.13) mm, rotated rx -9.61 ry -16.54 rz 125.97 deg; joints [-14.704, -58.39, 111.577, 191.498, 37.473, -112.334, -235]
  MoveL 2229 to (31.22, -49.73, -242.41) mm, rotated rx -9.61 ry -16.54 rz 125.97 deg; joints [-14.719, -58.316, 111.625, 191.444, 37.591, -112.28, -235]
  MoveL 2230 to (29.81, -50.98, -242.71) mm, rotated rx -9.61 ry -16.54 rz 125.97 deg; joints [-14.734, -58.245, 111.675, 191.389, 37.708, -112.226, -235]
  MoveL 2231 to (28.34, -52.33, -242.86) mm, rotated rx -9.61 ry -16.54 rz 125.97 deg; joints [-14.744, -58.169, 111.728, 191.341, 37.833, -112.176, -235]
  MoveL 2232 to (27.69, -52.32, -243.48) mm, rotated rx -9.61 ry -16.54 rz 125.97 deg; joints [-14.773, -58.171, 111.768, 191.286, 37.867, -112.136, -235]
  MoveL 2233 to (27.8, -52.02, -243.79) mm, rotated rx -9.61 ry -16.54 rz 125.97 deg; joints [-14.786, -58.188, 111.767, 191.271, 37.849, -112.129, -235]
  MoveL 2234 to (27.77, -51.98, -243.98) mm, rotated rx -9.61 ry -16.54 rz 125.97 deg; joints [-14.794, -58.189, 111.768, 191.258, 37.847, -112.122, -235]
  MoveL 2235 to (27.63, -52.19, -244.08) mm, rotated rx -9.61 ry -16.54 rz 125.97 deg; joints [-14.798, -58.176, 111.768, 191.249, 37.86, -112.114, -235]
  MoveL 2236 to (27.45, -52.6, -244.1) mm, rotated rx -9.61 ry -16.54 rz 125.97 deg; joints [-14.798, -58.15, 111.764, 191.243, 37.882, -112.107, -235]
  MoveL 2237 to (27.29, -53.06, -244.1) mm, rotated rx -9.61 ry -16.54 rz 125.97 deg; joints [-14.798, -58.12, 111.757, 191.238, 37.904, -112.1, -235]
  MoveL 2238 to (27.08, -54.01, -244.14) mm, rotated rx -9.61 ry -16.54 rz 125.97 deg; joints [-14.796, -58.058, 111.733, 191.231, 37.941, -112.089, -235]
  MoveL 2239 to (26.74, -55.55, -244.14) mm, rotated rx -9.61 ry -16.54 rz 125.97 deg; joints [-14.792, -57.958, 111.694, 191.222, 38.002, -112.074, -235]
  MoveL 2240 to (26.49, -56.5, -244.15) mm, rotated rx -9.61 ry -16.54 rz 125.97 deg; joints [-14.79, -57.896, 111.672, 191.215, 38.041, -112.063, -235]
  MoveL 2241 to (26.27, -57.52, -244.15) mm, rotated rx -9.61 ry -16.54 rz 125.97 deg; joints [-14.788, -57.829, 111.646, 191.209, 38.081, -112.053, -235]
  MoveL 2242 to (26.15, -58.02, -244.17) mm, rotated rx -9.61 ry -16.54 rz 125.97 deg; joints [-14.787, -57.796, 111.633, 191.205, 38.101, -112.047, -235]
  MoveL 2243 to (26.04, -58.48, -244.2) mm, rotated rx -9.61 ry -16.54 rz 125.97 deg; joints [-14.787, -57.767, 111.622, 191.2, 38.12, -112.041, -235]
  MoveL 2244 to (25.92, -58.9, -244.24) mm, rotated rx -9.61 ry -16.54 rz 125.97 deg; joints [-14.788, -57.739, 111.612, 191.194, 38.137, -112.035, -235]
  MoveL 2245 to (25.81, -59.29, -244.31) mm, rotated rx -9.61 ry -16.54 rz 125.97 deg; joints [-14.789, -57.713, 111.604, 191.188, 38.153, -112.028, -235]
  MoveL 2246 to (25.69, -59.69, -244.36) mm, rotated rx -9.61 ry -16.54 rz 125.97 deg; joints [-14.791, -57.687, 111.595, 191.182, 38.17, -112.021, -235]
  MoveL 2247 to (25.57, -60.14, -244.39) mm, rotated rx -9.61 ry -16.54 rz 125.97 deg; joints [-14.791, -57.658, 111.584, 191.177, 38.188, -112.015, -235]
  MoveL 2248 to (25.46, -60.6, -244.42) mm, rotated rx -9.61 ry -16.54 rz 125.97 deg; joints [-14.791, -57.627, 111.573, 191.172, 38.207, -112.009, -235]
  MoveL 2249 to (25.34, -61.02, -244.46) mm, rotated rx -9.61 ry -16.54 rz 125.97 deg; joints [-14.792, -57.6, 111.563, 191.167, 38.225, -112.003, -235]
  MoveL 2250 to (25.21, -61.41, -244.52) mm, rotated rx -9.61 ry -16.54 rz 125.97 deg; joints [-14.793, -57.575, 111.556, 191.16, 38.242, -111.996, -235]
  MoveL 2251 to (25.09, -61.8, -244.57) mm, rotated rx -9.61 ry -16.54 rz 125.97 deg; joints [-14.794, -57.549, 111.547, 191.154, 38.259, -111.99, -235]
  MoveL 2252 to (24.97, -62.22, -244.6) mm, rotated rx -9.61 ry -16.54 rz 125.97 deg; joints [-14.795, -57.521, 111.537, 191.149, 38.276, -111.984, -235]
  MoveL 2253 to (24.86, -62.73, -244.6) mm, rotated rx -9.61 ry -16.54 rz 125.97 deg; joints [-14.793, -57.488, 111.524, 191.146, 38.296, -111.979, -235]
  MoveL 2254 to (23.99, -65.52, -244.96) mm, rotated rx -9.61 ry -16.54 rz 125.97 deg; joints [-14.802, -57.306, 111.465, 191.103, 38.416, -111.933, -235]
  MoveL 2255 to (23.41, -66.67, -245.4) mm, rotated rx -9.61 ry -16.54 rz 125.97 deg; joints [-14.818, -57.23, 111.452, 191.063, 38.476, -111.898, -235]
  MoveL 2256 to (22.74, -67.66, -246.03) mm, rotated rx -9.61 ry -16.54 rz 125.97 deg; joints [-14.843, -57.164, 111.451, 191.009, 38.536, -111.855, -235]
  MoveL 2257 to (21.11, -69.17, -247.81) mm, rotated rx -9.61 ry -16.54 rz 125.97 deg; joints [-14.918, -57.064, 111.48, 190.863, 38.655, -111.747, -235]
  MoveL 2258 to (19.1, -70.04, -250.3) mm, rotated rx -9.61 ry -16.54 rz 125.97 deg; joints [-15.027, -57.003, 111.553, 190.666, 38.775, -111.607, -235]
  MoveL 2259 to (17.3, -70.14, -252.79) mm, rotated rx -9.61 ry -16.54 rz 125.97 deg; joints [-15.138, -56.991, 111.643, 190.475, 38.863, -111.477, -235]
  MoveL 2260 to (16.71, -69.87, -253.77) mm, rotated rx -9.61 ry -16.54 rz 125.97 deg; joints [-15.182, -57.008, 111.684, 190.402, 38.882, -111.43, -235]
  MoveL 2261 to (16.31, -69.36, -254.58) mm, rotated rx -9.61 ry -16.54 rz 125.97 deg; joints [-15.218, -57.038, 111.722, 190.345, 38.886, -111.395, -235]
  MoveL 2262 to (16.19, -69.03, -254.91) mm, rotated rx -9.61 ry -16.54 rz 125.97 deg; joints [-15.234, -57.059, 111.74, 190.321, 38.881, -111.382, -235]
  MoveL 2263 to (16.12, -68.64, -255.2) mm, rotated rx -9.61 ry -16.54 rz 125.97 deg; joints [-15.248, -57.084, 111.757, 190.302, 38.873, -111.371, -235]
  MoveL 2264 to (16.13, -67.69, -255.64) mm, rotated rx -9.61 ry -16.54 rz 125.97 deg; joints [-15.269, -57.144, 111.79, 190.275, 38.844, -111.359, -235]
  MoveL 2265 to (16.34, -66.52, -255.91) mm, rotated rx -9.61 ry -16.54 rz 125.97 deg; joints [-15.284, -57.219, 111.82, 190.263, 38.798, -111.359, -235]
  MoveL 2266 to (16.76, -65.13, -256) mm, rotated rx -9.61 ry -16.54 rz 125.97 deg; joints [-15.291, -57.308, 111.847, 190.267, 38.736, -111.37, -235]
  MoveL 2267 to (17.61, -62.66, -256) mm, rotated rx -9.61 ry -16.54 rz 125.97 deg; joints [-15.296, -57.468, 111.89, 190.285, 38.621, -111.399, -235]
  MoveL 2268 to (17.76, -62.25, -255.97) mm, rotated rx -9.61 ry -16.54 rz 125.97 deg; joints [-15.295, -57.494, 111.896, 190.29, 38.601, -111.405, -235]
  MoveL 2269 to (17.92, -61.87, -255.92) mm, rotated rx -9.61 ry -16.54 rz 125.97 deg; joints [-15.294, -57.518, 111.901, 190.296, 38.582, -111.412, -235]
  MoveL 2270 to (18.08, -61.52, -255.85) mm, rotated rx -9.61 ry -16.54 rz 125.97 deg; joints [-15.292, -57.541, 111.906, 190.304, 38.564, -111.42, -235]
  MoveL 2271 to (18.24, -61.12, -255.8) mm, rotated rx -9.61 ry -16.54 rz 125.97 deg; joints [-15.29, -57.567, 111.911, 190.311, 38.544, -111.427, -235]
  MoveL 2272 to (18.42, -60.66, -255.76) mm, rotated rx -9.61 ry -16.54 rz 125.97 deg; joints [-15.29, -57.597, 111.918, 190.317, 38.522, -111.434, -235]
  MoveL 2273 to (18.62, -60.17, -255.71) mm, rotated rx -9.61 ry -16.54 rz 125.97 deg; joints [-15.288, -57.629, 111.925, 190.325, 38.497, -111.442, -235]
  MoveL 2274 to (18.81, -59.66, -255.69) mm, rotated rx -9.61 ry -16.54 rz 125.97 deg; joints [-15.288, -57.661, 111.933, 190.33, 38.473, -111.449, -235]
  MoveL 2275 to (19.01, -59.05, -255.7) mm, rotated rx -9.61 ry -16.54 rz 125.97 deg; joints [-15.29, -57.7, 111.943, 190.333, 38.444, -111.456, -235]
  MoveL 2276 to (19.27, -58.22, -255.77) mm, rotated rx -9.61 ry -16.54 rz 125.97 deg; joints [-15.295, -57.754, 111.958, 190.335, 38.406, -111.463, -235]
  MoveL 2277 to (19.44, -57.72, -255.77) mm, rotated rx -9.61 ry -16.54 rz 125.97 deg; joints [-15.296, -57.785, 111.966, 190.339, 38.383, -111.468, -235]
  MoveL 2278 to (19.6, -57.25, -255.76) mm, rotated rx -9.61 ry -16.54 rz 125.97 deg; joints [-15.297, -57.816, 111.974, 190.343, 38.361, -111.474, -235]
  MoveL 2279 to (19.76, -56.82, -255.74) mm, rotated rx -9.61 ry -16.54 rz 125.97 deg; joints [-15.297, -57.844, 111.981, 190.348, 38.34, -111.481, -235]
  MoveL 2280 to (19.92, -56.43, -255.69) mm, rotated rx -9.61 ry -16.54 rz 125.97 deg; joints [-15.295, -57.869, 111.985, 190.354, 38.32, -111.488, -235]
  MoveL 2281 to (20.09, -56.07, -255.63) mm, rotated rx -9.61 ry -16.54 rz 125.97 deg; joints [-15.293, -57.892, 111.989, 190.362, 38.301, -111.495, -235]
  MoveL 2282 to (20.31, -55.71, -255.58) mm, rotated rx -9.61 ry -16.54 rz 125.97 deg; joints [-15.291, -57.914, 111.988, 190.37, 38.279, -111.504, -235]
  MoveL 2283 to (20.56, -55.39, -255.52) mm, rotated rx -9.61 ry -16.54 rz 125.97 deg; joints [-15.289, -57.935, 111.984, 190.379, 38.255, -111.513, -235]
  MoveL 2284 to (20.74, -55.25, -255.36) mm, rotated rx -9.61 ry -16.54 rz 125.97 deg; joints [-15.282, -57.943, 111.979, 190.394, 38.242, -111.524, -235]
  MoveL 2285 to (20.74, -55.36, -255.05) mm, rotated rx -9.61 ry -16.54 rz 125.97 deg; joints [-15.269, -57.939, 111.979, 190.413, 38.248, -111.534, -235]
  MoveL 2286 to (20.54, -55.75, -254.56) mm, rotated rx -9.61 ry -16.54 rz 125.97 deg; joints [-15.249, -57.919, 111.987, 190.437, 38.277, -111.545, -235]
  MoveL 2287 to (21.22, -55.18, -253.71) mm, rotated rx -9.61 ry -16.54 rz 125.97 deg; joints [-15.212, -57.957, 111.973, 190.505, 38.229, -111.594, -235]
  MoveL 2288 to (24.62, -52.6, -253.71) mm, rotated rx -9.61 ry -16.54 rz 125.97 deg; joints [-15.202, -58.097, 111.825, 190.589, 37.948, -111.689, -235]
  MoveL 2289 to (26.22, -51.39, -253.64) mm, rotated rx -9.61 ry -16.54 rz 125.97 deg; joints [-15.194, -58.162, 111.756, 190.632, 37.817, -111.737, -235]
  MoveL 2290 to (27.81, -50.2, -253.49) mm, rotated rx -9.61 ry -16.54 rz 125.97 deg; joints [-15.183, -58.227, 111.688, 190.681, 37.687, -111.788, -235]
  MoveL 2291 to (29.65, -48.83, -253.3) mm, rotated rx -9.61 ry -16.54 rz 125.97 deg; joints [-15.17, -58.301, 111.609, 190.739, 37.538, -111.847, -235]
  MoveL 2292 to (31.39, -47.53, -253.08) mm, rotated rx -9.61 ry -16.54 rz 125.97 deg; joints [-15.156, -58.371, 111.534, 190.797, 37.397, -111.905, -235]
  MoveL 2293 to (33.13, -46.22, -252.98) mm, rotated rx -9.61 ry -16.54 rz 125.97 deg; joints [-15.146, -58.441, 111.458, 190.848, 37.255, -111.96, -235]
  MoveL 2294 to (34.83, -44.93, -252.98) mm, rotated rx -9.61 ry -16.54 rz 125.97 deg; joints [-15.141, -58.509, 111.382, 190.892, 37.114, -112.01, -235]
  MoveL 2295 to (36.41, -43.72, -252.92) mm, rotated rx -9.61 ry -16.54 rz 125.97 deg; joints [-15.134, -58.572, 111.312, 190.937, 36.984, -112.059, -235]
  MoveL 2296 to (37.9, -42.58, -252.8) mm, rotated rx -9.61 ry -16.54 rz 125.97 deg; joints [-15.124, -58.633, 111.247, 190.983, 36.862, -112.108, -235]
  MoveL 2297 to (39.53, -41.35, -252.73) mm, rotated rx -9.61 ry -16.54 rz 125.97 deg; joints [-15.117, -58.697, 111.174, 191.03, 36.729, -112.159, -235]
  MoveL 2298 to (41.22, -40.05, -252.55) mm, rotated rx -9.61 ry -16.54 rz 125.97 deg; joints [-15.104, -58.765, 111.1, 191.087, 36.591, -112.217, -235]
  MoveL 2299 to (44.62, -37.46, -252.37) mm, rotated rx -9.61 ry -16.54 rz 125.97 deg; joints [-15.087, -58.899, 110.948, 191.19, 36.312, -112.328, -235]
  MoveL 2300 to (46.31, -36.16, -252.19) mm, rotated rx -9.61 ry -16.54 rz 125.97 deg; joints [-15.074, -58.967, 110.873, 191.247, 36.174, -112.387, -235]
  MoveL 2301 to (48, -34.85, -252.01) mm, rotated rx -9.61 ry -16.54 rz 125.97 deg; joints [-15.062, -59.034, 110.799, 191.305, 36.036, -112.447, -235]
  MoveL 2302 to (49.7, -33.56, -252.01) mm, rotated rx -9.61 ry -16.54 rz 125.97 deg; joints [-15.057, -59.099, 110.72, 191.352, 35.896, -112.501, -235]
  MoveL 2303 to (51.38, -32.25, -251.83) mm, rotated rx -9.61 ry -16.54 rz 125.97 deg; joints [-15.045, -59.166, 110.645, 191.411, 35.758, -112.561, -235]
  MoveL 2304 to (53.06, -30.94, -251.66) mm, rotated rx -9.61 ry -16.54 rz 125.97 deg; joints [-15.033, -59.233, 110.57, 191.47, 35.62, -112.622, -235]
  MoveL 2305 to (54.76, -29.65, -251.66) mm, rotated rx -9.61 ry -16.54 rz 125.97 deg; joints [-15.028, -59.297, 110.49, 191.518, 35.48, -112.677, -235]
  MoveL 2306 to (56.27, -28.41, -251.46) mm, rotated rx -9.61 ry -16.54 rz 125.97 deg; joints [-15.016, -59.361, 110.425, 191.574, 35.355, -112.734, -235]
  MoveL 2307 to (57.55, -27.27, -251.14) mm, rotated rx -9.61 ry -16.54 rz 125.97 deg; joints [-15, -59.422, 110.376, 191.632, 35.249, -112.789, -235]
  MoveL 2308 to (58.64, -26.2, -250.68) mm, rotated rx -9.61 ry -16.54 rz 125.97 deg; joints [-14.979, -59.483, 110.341, 191.693, 35.158, -112.845, -235]
  MoveL 2309 to (57.79, -26.63, -249.91) mm, rotated rx -9.61 ry -16.54 rz 125.97 deg; joints [-14.952, -59.473, 110.402, 191.718, 35.231, -112.849, -235]
  MoveL 2310 to (58.15, -26.41, -249.9) mm, rotated rx -9.61 ry -16.54 rz 125.97 deg; joints [-14.95, -59.482, 110.383, 191.729, 35.204, -112.861, -235]
  MoveC 2311 to (61.66, -25.91, -249.9) mm, rotated rx -9.61 ry -16.54 rz 125.97 deg; joints [-14.931, -59.467, 110.129, 191.83, 34.972, -112.967, -235] to (65.21, -25.71, -249.9) mm, rotated rx -9.61 ry -16.54 rz 125.97 deg; joints [-14.91, -59.43, 109.859, 191.934, 34.747, -113.073, -235]
  MoveL 2312 to (65.21, -25.71, -249.9) mm, rotated rx -9.61 ry -16.54 rz 125.97 deg; joints [-14.91, -59.43, 109.859, 191.934, 34.747, -113.073, -235]
  MoveL 2313 to (65.68, -25.67, -249.88) mm, rotated rx -9.61 ry -16.54 rz 125.97 deg; joints [-14.907, -59.426, 109.825, 191.949, 34.717, -113.088, -235]
  MoveL 2314 to (66.1, -25.62, -249.83) mm, rotated rx -9.61 ry -16.54 rz 125.97 deg; joints [-14.902, -59.425, 109.795, 191.964, 34.691, -113.103, -235]
  MoveL 2315 to (66.5, -25.56, -249.77) mm, rotated rx -9.61 ry -16.54 rz 125.97 deg; joints [-14.898, -59.423, 109.767, 191.98, 34.665, -113.118, -235]
  MoveL 2316 to (66.94, -25.51, -249.72) mm, rotated rx -9.61 ry -16.54 rz 125.97 deg; joints [-14.893, -59.421, 109.735, 191.996, 34.637, -113.133, -235]
  MoveL 2317 to (67.41, -25.46, -249.7) mm, rotated rx -9.61 ry -16.54 rz 125.97 deg; joints [-14.89, -59.417, 109.7, 192.012, 34.607, -113.149, -235]
  MoveL 2318 to (67.93, -25.43, -249.68) mm, rotated rx -9.61 ry -16.54 rz 125.97 deg; joints [-14.886, -59.412, 109.662, 192.028, 34.575, -113.165, -235]
  MoveL 2319 to (68.97, -25.36, -249.68) mm, rotated rx -9.61 ry -16.54 rz 125.97 deg; joints [-14.88, -59.401, 109.582, 192.059, 34.508, -113.197, -235]
  MoveL 2320 to (70.43, -25.33, -249.77) mm, rotated rx -9.61 ry -16.54 rz 125.97 deg; joints [-14.875, -59.381, 109.467, 192.096, 34.416, -113.238, -235]
  MoveL 2321 to (71.62, -25.43, -250.05) mm, rotated rx -9.61 ry -16.54 rz 125.97 deg; joints [-14.878, -59.355, 109.365, 192.114, 34.342, -113.262, -235]
  MoveL 2322 to (72.56, -25.67, -250.5) mm, rotated rx -9.61 ry -16.54 rz 125.97 deg; joints [-14.89, -59.322, 109.275, 192.112, 34.285, -113.271, -235]
  MoveL 2323 to (73.24, -26.03, -251.14) mm, rotated rx -9.61 ry -16.54 rz 125.97 deg; joints [-14.91, -59.282, 109.197, 192.09, 34.244, -113.263, -235]
  MoveL 2324 to (73.67, -26.52, -251.97) mm, rotated rx -9.61 ry -16.54 rz 125.97 deg; joints [-14.938, -59.236, 109.131, 192.049, 34.221, -113.239, -235]
  MoveL 2325 to (73.83, -27.14, -252.97) mm, rotated rx -9.61 ry -16.54 rz 125.97 deg; joints [-14.974, -59.183, 109.077, 191.988, 34.215, -113.198, -235]
  MoveL 2326 to (73.39, -28.77, -255.53) mm, rotated rx -9.61 ry -16.54 rz 125.97 deg; joints [-15.071, -59.059, 109.007, 191.807, 34.255, -113.07, -235]
  MoveL 2327 to (72.15, -30.4, -258.09) mm, rotated rx -9.61 ry -16.54 rz 125.97 deg; joints [-15.173, -58.946, 108.997, 191.604, 34.343, -112.918, -235]
  MoveL 2328 to (71.32, -31.03, -259.1) mm, rotated rx -9.61 ry -16.54 rz 125.97 deg; joints [-15.215, -58.907, 109.021, 191.515, 34.399, -112.849, -235]
  MoveL 2329 to (70.36, -31.53, -259.92) mm, rotated rx -9.61 ry -16.54 rz 125.97 deg; joints [-15.252, -58.881, 109.063, 191.434, 34.462, -112.785, -235]
  MoveL 2330 to (69.26, -31.9, -260.56) mm, rotated rx -9.61 ry -16.54 rz 125.97 deg; joints [-15.282, -58.866, 109.124, 191.36, 34.532, -112.724, -235]
  MoveL 2331 to (68.01, -32.14, -261.02) mm, rotated rx -9.61 ry -16.54 rz 125.97 deg; joints [-15.307, -58.864, 109.204, 191.295, 34.61, -112.669, -235]
  MoveL 2332 to (65.12, -32.24, -261.38) mm, rotated rx -9.61 ry -16.54 rz 125.97 deg; joints [-15.339, -58.894, 109.421, 191.189, 34.788, -112.57, -235]
  MoveL 2333 to (64.07, -32.19, -261.38) mm, rotated rx -9.61 ry -16.54 rz 125.97 deg; joints [-15.346, -58.912, 109.505, 191.159, 34.852, -112.54, -235]
  MoveL 2334 to (63.55, -32.17, -261.39) mm, rotated rx -9.61 ry -16.54 rz 125.97 deg; joints [-15.35, -58.921, 109.546, 191.144, 34.884, -112.525, -235]
  MoveL 2335 to (63.07, -32.16, -261.41) mm, rotated rx -9.61 ry -16.54 rz 125.97 deg; joints [-15.354, -58.928, 109.583, 191.129, 34.913, -112.51, -235]
  MoveL 2336 to (62.65, -32.17, -261.46) mm, rotated rx -9.61 ry -16.54 rz 125.97 deg; joints [-15.358, -58.933, 109.616, 191.114, 34.939, -112.496, -235]
  MoveL 2337 to (62.25, -32.18, -261.52) mm, rotated rx -9.61 ry -16.54 rz 125.97 deg; joints [-15.363, -58.937, 109.646, 191.099, 34.963, -112.483, -235]
  MoveL 2338 to (61.83, -32.18, -261.56) mm, rotated rx -9.61 ry -16.54 rz 125.97 deg; joints [-15.367, -58.942, 109.677, 191.084, 34.989, -112.469, -235]
  MoveL 2339 to (61.36, -32.17, -261.59) mm, rotated rx -9.61 ry -16.54 rz 125.97 deg; joints [-15.371, -58.949, 109.714, 191.07, 35.018, -112.455, -235]
  MoveL 2340 to (60.86, -32.15, -261.59) mm, rotated rx -9.61 ry -16.54 rz 125.97 deg; joints [-15.375, -58.957, 109.753, 191.056, 35.048, -112.44, -235]
  MoveL 2341 to (60.31, -32.12, -261.59) mm, rotated rx -9.61 ry -16.54 rz 125.97 deg; joints [-15.378, -58.967, 109.798, 191.041, 35.082, -112.425, -235]
  MoveL 2342 to (59.78, -32.1, -261.59) mm, rotated rx -9.61 ry -16.54 rz 125.97 deg; joints [-15.382, -58.976, 109.84, 191.025, 35.114, -112.41, -235]
  MoveL 2343 to (59.29, -32.09, -261.62) mm, rotated rx -9.61 ry -16.54 rz 125.97 deg; joints [-15.386, -58.983, 109.878, 191.01, 35.144, -112.395, -235]
  MoveL 2344 to (58.81, -32.08, -261.66) mm, rotated rx -9.61 ry -16.54 rz 125.97 deg; joints [-15.391, -58.989, 109.914, 190.994, 35.173, -112.38, -235]
  MoveL 2345 to (58.31, -32.1, -261.74) mm, rotated rx -9.61 ry -16.54 rz 125.97 deg; joints [-15.397, -58.995, 109.952, 190.975, 35.204, -112.363, -235]
  MoveL 2346 to (57.7, -32.11, -261.8) mm, rotated rx -9.61 ry -16.54 rz 125.97 deg; joints [-15.403, -59.002, 109.997, 190.954, 35.241, -112.343, -235]
  MoveL 2347 to (57.13, -32.09, -261.82) mm, rotated rx -9.61 ry -16.54 rz 125.97 deg; joints [-15.408, -59.01, 110.042, 190.937, 35.276, -112.327, -235]
  MoveL 2348 to (56.61, -32.07, -261.82) mm, rotated rx -9.61 ry -16.54 rz 125.97 deg; joints [-15.411, -59.019, 110.084, 190.922, 35.308, -112.312, -235]
  MoveL 2349 to (56.08, -32.04, -261.82) mm, rotated rx -9.61 ry -16.54 rz 125.97 deg; joints [-15.415, -59.027, 110.125, 190.908, 35.34, -112.298, -235]
  MoveL 2350 to (55.42, -32.03, -261.83) mm, rotated rx -9.61 ry -16.54 rz 125.97 deg; joints [-15.419, -59.037, 110.177, 190.889, 35.381, -112.279, -235]
  MoveL 2351 to (54.84, -32.04, -261.84) mm, rotated rx -9.61 ry -16.54 rz 125.97 deg; joints [-15.423, -59.044, 110.222, 190.873, 35.417, -112.262, -235]
  MoveL 2352 to (54.33, -32.07, -261.85) mm, rotated rx -9.61 ry -16.54 rz 125.97 deg; joints [-15.427, -59.048, 110.259, 190.858, 35.449, -112.248, -235]
  MoveL 2353 to (54, -32.15, -261.85) mm, rotated rx -9.61 ry -16.54 rz 125.97 deg; joints [-15.429, -59.048, 110.282, 190.849, 35.472, -112.238, -235]
  MoveL 2354 to (53.75, -32.25, -261.85) mm, rotated rx -9.61 ry -16.54 rz 125.97 deg; joints [-15.43, -59.044, 110.298, 190.842, 35.491, -112.231, -235]
  MoveL 2355 to (54.61, -31.88, -262.44) mm, rotated rx -9.61 ry -16.54 rz 125.97 deg; joints [-15.449, -59.052, 110.235, 190.828, 35.42, -112.233, -235]
  MoveL 2356 to (53.63, -32.79, -262.97) mm, rotated rx -9.61 ry -16.54 rz 125.97 deg; joints [-15.473, -58.999, 110.266, 190.768, 35.499, -112.181, -235]
  MoveL 2357 to (52.4, -33.75, -263.35) mm, rotated rx -9.61 ry -16.54 rz 125.97 deg; joints [-15.492, -58.948, 110.317, 190.71, 35.597, -112.128, -235]
  MoveL 2358 to (50.87, -34.78, -263.61) mm, rotated rx -9.61 ry -16.54 rz 125.97 deg; joints [-15.507, -58.897, 110.389, 190.653, 35.716, -112.073, -235]
  MoveL 2359 to (49.13, -35.87, -263.74) mm, rotated rx -9.61 ry -16.54 rz 125.97 deg; joints [-15.519, -58.846, 110.478, 190.598, 35.853, -112.017, -235]
  MoveL 2360 to (47.33, -36.97, -263.83) mm, rotated rx -9.61 ry -16.54 rz 125.97 deg; joints [-15.529, -58.794, 110.57, 190.545, 35.993, -111.961, -235]
  MoveL 2361 to (43.69, -39.18, -264.01) mm, rotated rx -9.61 ry -16.54 rz 125.97 deg; joints [-15.55, -58.69, 110.758, 190.438, 36.277, -111.849, -235]
  MoveL 2362 to (41.87, -40.3, -264.19) mm, rotated rx -9.61 ry -16.54 rz 125.97 deg; joints [-15.564, -58.636, 110.849, 190.38, 36.419, -111.79, -235]
  MoveL 2363 to (38.22, -42.51, -264.37) mm, rotated rx -9.61 ry -16.54 rz 125.97 deg; joints [-15.586, -58.53, 111.035, 190.275, 36.704, -111.681, -235]
  MoveL 2364 to (36.39, -43.61, -264.55) mm, rotated rx -9.61 ry -16.54 rz 125.97 deg; joints [-15.6, -58.475, 111.126, 190.218, 36.845, -111.624, -235]
  MoveL 2365 to (34.56, -44.71, -264.64) mm, rotated rx -9.61 ry -16.54 rz 125.97 deg; joints [-15.611, -58.422, 111.218, 190.166, 36.988, -111.57, -235]
  MoveL 2366 to (32.86, -45.71, -264.86) mm, rotated rx -9.61 ry -16.54 rz 125.97 deg; joints [-15.626, -58.372, 111.303, 190.111, 37.119, -111.516, -235]
  MoveL 2367 to (30.84, -46.93, -265) mm, rotated rx -9.61 ry -16.54 rz 125.97 deg; joints [-15.639, -58.311, 111.404, 190.052, 37.276, -111.456, -235]
  MoveL 2368 to (28.64, -48.25, -265.12) mm, rotated rx -9.61 ry -16.54 rz 125.97 deg; joints [-15.653, -58.245, 111.513, 189.991, 37.447, -111.392, -235]
  MoveL 2369 to (26.82, -49.35, -265.12) mm, rotated rx -9.61 ry -16.54 rz 125.97 deg; joints [-15.66, -58.191, 111.606, 189.947, 37.591, -111.344, -235]
  MoveL 2370 to (25.07, -50.39, -265.2) mm, rotated rx -9.61 ry -16.54 rz 125.97 deg; joints [-15.67, -58.139, 111.693, 189.9, 37.728, -111.295, -235]
  MoveL 2371 to (23.49, -51.32, -265.37) mm, rotated rx -9.61 ry -16.54 rz 125.97 deg; joints [-15.683, -58.091, 111.771, 189.852, 37.85, -111.247, -235]
  MoveL 2372 to (21.87, -52.25, -265.58) mm, rotated rx -9.61 ry -16.54 rz 125.97 deg; joints [-15.698, -58.043, 111.85, 189.801, 37.974, -111.198, -235]
  MoveL 2373 to (19.84, -53.45, -265.72) mm, rotated rx -9.61 ry -16.54 rz 125.97 deg; joints [-15.711, -57.981, 111.95, 189.745, 38.132, -111.14, -235]
  MoveL 2374 to (17.63, -54.77, -265.82) mm, rotated rx -9.61 ry -16.54 rz 125.97 deg; joints [-15.724, -57.913, 112.059, 189.687, 38.305, -111.08, -235]
  MoveL 2375 to (13.97, -56.97, -265.82) mm, rotated rx -9.61 ry -16.54 rz 125.97 deg; joints [-15.739, -57.8, 112.24, 189.603, 38.594, -110.988, -235]
  MoveL 2376 to (13.67, -56.88, -266.52) mm, rotated rx -9.61 ry -16.54 rz 125.97 deg; joints [-15.769, -57.802, 112.254, 189.554, 38.602, -110.956, -235]
  MoveL 2377 to (13.85, -56.63, -266.86) mm, rotated rx -9.61 ry -16.54 rz 125.97 deg; joints [-15.783, -57.815, 112.245, 189.537, 38.58, -110.949, -235]
  MoveL 2378 to (13.84, -56.61, -267.08) mm, rotated rx -9.61 ry -16.54 rz 125.97 deg; joints [-15.792, -57.814, 112.243, 189.524, 38.578, -110.942, -235]
  MoveL 2379 to (13.67, -56.82, -267.19) mm, rotated rx -9.61 ry -16.54 rz 125.97 deg; joints [-15.796, -57.801, 112.245, 189.513, 38.592, -110.933, -235]
  MoveL 2380 to (13.43, -57.2, -267.22) mm, rotated rx -9.61 ry -16.54 rz 125.97 deg; joints [-15.798, -57.777, 112.247, 189.506, 38.617, -110.925, -235]
  MoveL 2381 to (13.19, -57.61, -267.25) mm, rotated rx -9.61 ry -16.54 rz 125.97 deg; joints [-15.798, -57.751, 112.246, 189.5, 38.642, -110.918, -235]
  MoveL 2382 to (12.99, -57.99, -267.3) mm, rotated rx -9.61 ry -16.54 rz 125.97 deg; joints [-15.8, -57.727, 112.245, 189.493, 38.665, -110.911, -235]
  MoveL 2383 to (12.79, -58.34, -267.37) mm, rotated rx -9.61 ry -16.54 rz 125.97 deg; joints [-15.802, -57.704, 112.244, 189.485, 38.685, -110.903, -235]
  MoveL 2384 to (12.59, -58.7, -267.42) mm, rotated rx -9.61 ry -16.54 rz 125.97 deg; joints [-15.804, -57.681, 112.242, 189.477, 38.706, -110.895, -235]
  MoveL 2385 to (12.38, -59.09, -267.46) mm, rotated rx -9.61 ry -16.54 rz 125.97 deg; joints [-15.806, -57.656, 112.24, 189.471, 38.729, -110.888, -235]
  MoveL 2386 to (12.15, -59.56, -267.49) mm, rotated rx -9.61 ry -16.54 rz 125.97 deg; joints [-15.806, -57.627, 112.237, 189.464, 38.756, -110.881, -235]
  MoveL 2387 to (11.9, -60.03, -267.55) mm, rotated rx -9.61 ry -16.54 rz 125.97 deg; joints [-15.808, -57.597, 112.235, 189.455, 38.783, -110.871, -235]
  MoveL 2388 to (11.66, -60.49, -267.58) mm, rotated rx -9.61 ry -16.54 rz 125.97 deg; joints [-15.809, -57.567, 112.233, 189.449, 38.809, -110.864, -235]
  MoveL 2389 to (11.44, -60.96, -267.59) mm, rotated rx -9.61 ry -16.54 rz 125.97 deg; joints [-15.809, -57.537, 112.229, 189.444, 38.835, -110.857, -235]
  MoveL 2390 to (11.22, -61.44, -267.59) mm, rotated rx -9.61 ry -16.54 rz 125.97 deg; joints [-15.808, -57.507, 112.225, 189.44, 38.861, -110.851, -235]
  MoveL 2391 to (10.94, -62.07, -267.55) mm, rotated rx -9.61 ry -16.54 rz 125.97 deg; joints [-15.806, -57.467, 112.22, 189.436, 38.895, -110.844, -235]
  MoveL 2392 to (10.67, -62.67, -267.52) mm, rotated rx -9.61 ry -16.54 rz 125.97 deg; joints [-15.803, -57.429, 112.214, 189.433, 38.928, -110.837, -235]
  MoveL 2393 to (10.42, -63.22, -267.52) mm, rotated rx -9.61 ry -16.54 rz 125.97 deg; joints [-15.802, -57.394, 112.21, 189.428, 38.958, -110.83, -235]
  MoveL 2394 to (10.2, -63.63, -267.55) mm, rotated rx -9.61 ry -16.54 rz 125.97 deg; joints [-15.803, -57.368, 112.207, 189.422, 38.981, -110.823, -235]
  MoveL 2395 to (10, -63.99, -267.61) mm, rotated rx -9.61 ry -16.54 rz 125.97 deg; joints [-15.806, -57.345, 112.206, 189.414, 39.003, -110.816, -235]
  MoveL 2396 to (9.8, -64.35, -267.67) mm, rotated rx -9.61 ry -16.54 rz 125.97 deg; joints [-15.807, -57.322, 112.204, 189.407, 39.024, -110.808, -235]
  MoveL 2397 to (9.6, -64.74, -267.7) mm, rotated rx -9.61 ry -16.54 rz 125.97 deg; joints [-15.808, -57.297, 112.202, 189.401, 39.046, -110.801, -235]
  MoveL 2398 to (8.93, -66.17, -267.7) mm, rotated rx -9.61 ry -16.54 rz 125.97 deg; joints [-15.807, -57.206, 112.191, 189.388, 39.124, -110.783, -235]
  MoveL 2399 to (7.5, -68.68, -268.08) mm, rotated rx -9.61 ry -16.54 rz 125.97 deg; joints [-15.82, -57.045, 112.182, 189.337, 39.273, -110.732, -235]
  MoveL 2400 to (6.72, -69.66, -268.55) mm, rotated rx -9.61 ry -16.54 rz 125.97 deg; joints [-15.84, -56.981, 112.189, 189.294, 39.341, -110.696, -235]
  MoveL 2401 to (5.91, -70.46, -269.21) mm, rotated rx -9.61 ry -16.54 rz 125.97 deg; joints [-15.868, -56.927, 112.203, 189.238, 39.406, -110.654, -235]
  MoveL 2402 to (5.05, -71.09, -270.06) mm, rotated rx -9.61 ry -16.54 rz 125.97 deg; joints [-15.905, -56.885, 112.225, 189.17, 39.466, -110.605, -235]
  MoveL 2403 to (4.15, -71.52, -271.09) mm, rotated rx -9.61 ry -16.54 rz 125.97 deg; joints [-15.95, -56.853, 112.254, 189.089, 39.522, -110.549, -235]
  MoveL 2404 to (2.23, -71.86, -273.73) mm, rotated rx -9.61 ry -16.54 rz 125.97 deg; joints [-16.068, -56.822, 112.335, 188.892, 39.622, -110.419, -235]
  MoveL 2405 to (0.69, -71.49, -276.37) mm, rotated rx -9.61 ry -16.54 rz 125.97 deg; joints [-16.186, -56.836, 112.419, 188.702, 39.682, -110.298, -235]
  MoveL 2406 to (0.25, -71.06, -277.4) mm, rotated rx -9.61 ry -16.54 rz 125.97 deg; joints [-16.232, -56.859, 112.452, 188.631, 39.687, -110.256, -235]
  MoveL 2407 to (0.05, -70.45, -278.25) mm, rotated rx -9.61 ry -16.54 rz 125.97 deg; joints [-16.27, -56.894, 112.478, 188.575, 39.675, -110.224, -235]
  MoveL 2408 to (0.07, -69.68, -278.91) mm, rotated rx -9.61 ry -16.54 rz 125.97 deg; joints [-16.3, -56.94, 112.498, 188.535, 39.647, -110.204, -235]
  MoveL 2409 to (0.32, -68.74, -279.38) mm, rotated rx -9.61 ry -16.54 rz 125.97 deg; joints [-16.322, -56.997, 112.512, 188.51, 39.603, -110.195, -235]
  MoveL 2410 to (0.79, -67.63, -279.66) mm, rotated rx -9.61 ry -16.54 rz 125.97 deg; joints [-16.335, -57.066, 112.52, 188.501, 39.541, -110.197, -235]
  MoveL 2411 to (1.5, -66.36, -279.76) mm, rotated rx -9.61 ry -16.54 rz 125.97 deg; joints [-16.34, -57.146, 112.522, 188.507, 39.463, -110.211, -235]
  MoveL 2412 to (1.77, -65.91, -279.76) mm, rotated rx -9.61 ry -16.54 rz 125.97 deg; joints [-16.34, -57.174, 112.522, 188.512, 39.435, -110.218, -235]
  MoveL 2413 to (2.02, -65.51, -279.74) mm, rotated rx -9.61 ry -16.54 rz 125.97 deg; joints [-16.34, -57.199, 112.521, 188.518, 39.409, -110.224, -235]
  MoveL 2414 to (2.25, -65.18, -279.69) mm, rotated rx -9.61 ry -16.54 rz 125.97 deg; joints [-16.338, -57.22, 112.519, 188.525, 39.387, -110.232, -235]
  MoveL 2415 to (2.47, -64.86, -279.63) mm, rotated rx -9.61 ry -16.54 rz 125.97 deg; joints [-16.335, -57.241, 112.517, 188.533, 39.365, -110.239, -235]
  MoveL 2416 to (2.71, -64.5, -279.59) mm, rotated rx -9.61 ry -16.54 rz 125.97 deg; joints [-16.334, -57.263, 112.515, 188.539, 39.341, -110.246, -235]
  MoveL 2417 to (2.98, -64.09, -279.57) mm, rotated rx -9.61 ry -16.54 rz 125.97 deg; joints [-16.333, -57.289, 112.514, 188.546, 39.314, -110.253, -235]
  MoveL 2418 to (3.25, -63.64, -279.57) mm, rotated rx -9.61 ry -16.54 rz 125.97 deg; joints [-16.333, -57.318, 112.513, 188.551, 39.286, -110.26, -235]
  MoveL 2419 to (3.49, -63.24, -279.54) mm, rotated rx -9.61 ry -16.54 rz 125.97 deg; joints [-16.332, -57.343, 112.512, 188.556, 39.26, -110.266, -235]
  MoveL 2420 to (3.72, -62.91, -279.49) mm, rotated rx -9.61 ry -16.54 rz 125.97 deg; joints [-16.33, -57.364, 112.511, 188.564, 39.238, -110.274, -235]
  MoveL 2421 to (3.93, -62.58, -279.43) mm, rotated rx -9.61 ry -16.54 rz 125.97 deg; joints [-16.328, -57.385, 112.51, 188.571, 39.217, -110.281, -235]
  MoveL 2422 to (4.17, -62.22, -279.39) mm, rotated rx -9.61 ry -16.54 rz 125.97 deg; joints [-16.326, -57.408, 112.509, 188.578, 39.193, -110.288, -235]
  MoveL 2423 to (4.43, -61.8, -279.36) mm, rotated rx -9.61 ry -16.54 rz 125.97 deg; joints [-16.325, -57.434, 112.508, 188.585, 39.167, -110.295, -235]
  MoveL 2424 to (4.7, -61.35, -279.36) mm, rotated rx -9.61 ry -16.54 rz 125.97 deg; joints [-16.326, -57.462, 112.508, 188.59, 39.138, -110.302, -235]
  MoveL 2425 to (5.27, -60.55, -279.34) mm, rotated rx -9.61 ry -16.54 rz 125.97 deg; joints [-16.325, -57.512, 112.5, 188.602, 39.081, -110.316, -235]
  MoveC 2426 to (6.09, -59.44, -279.34) mm, rotated rx -9.61 ry -16.54 rz 125.97 deg; joints [-16.324, -57.58, 112.486, 188.617, 39.001, -110.336, -235] to (6.78, -58.24, -279.34) mm, rotated rx -9.61 ry -16.54 rz 125.97 deg; joints [-16.325, -57.655, 112.486, 188.63, 38.927, -110.353, -235]
  MoveL 2427 to (6.78, -58.24, -279.33) mm, rotated rx -9.61 ry -16.54 rz 125.97 deg; joints [-16.325, -57.655, 112.486, 188.631, 38.927, -110.354, -235]
  MoveL 2428 to (7.15, -57.7, -279.32) mm, rotated rx -9.61 ry -16.54 rz 125.97 deg; joints [-16.324, -57.688, 112.482, 188.639, 38.889, -110.363, -235]
  MoveL 2429 to (7.52, -57.26, -279.29) mm, rotated rx -9.61 ry -16.54 rz 125.97 deg; joints [-16.322, -57.715, 112.473, 188.648, 38.854, -110.373, -235]
  MoveL 2430 to (7.77, -57.08, -279.19) mm, rotated rx -9.61 ry -16.54 rz 125.97 deg; joints [-16.318, -57.726, 112.465, 188.659, 38.835, -110.382, -235]
  MoveL 2431 to (7.76, -57.15, -278.99) mm, rotated rx -9.61 ry -16.54 rz 125.97 deg; joints [-16.309, -57.723, 112.466, 188.67, 38.84, -110.389, -235]
  MoveL 2432 to (7.48, -57.46, -278.69) mm, rotated rx -9.61 ry -16.54 rz 125.97 deg; joints [-16.297, -57.707, 112.479, 188.683, 38.869, -110.393, -235]
  MoveL 2433 to (7.58, -57.84, -278.06) mm, rotated rx -9.61 ry -16.54 rz 125.97 deg; joints [-16.27, -57.687, 112.466, 188.724, 38.879, -110.416, -235]
  MoveL 2434 to (9.38, -56.87, -278.06) mm, rotated rx -9.61 ry -16.54 rz 125.97 deg; joints [-16.262, -57.736, 112.374, 188.763, 38.74, -110.458, -235]
  MoveL 2435 to (11.31, -55.94, -278) mm, rotated rx -9.61 ry -16.54 rz 125.97 deg; joints [-16.251, -57.782, 112.271, 188.808, 38.594, -110.504, -235]
  MoveL 2436 to (13.37, -54.98, -277.88) mm, rotated rx -9.61 ry -16.54 rz 125.97 deg; joints [-16.236, -57.828, 112.159, 188.861, 38.44, -110.557, -235]
  MoveL 2437 to (15.4, -54.04, -277.78) mm, rotated rx -9.61 ry -16.54 rz 125.97 deg; joints [-16.222, -57.873, 112.049, 188.913, 38.288, -110.608, -235]
  MoveL 2438 to (17.35, -53.14, -277.6) mm, rotated rx -9.61 ry -16.54 rz 125.97 deg; joints [-16.206, -57.916, 111.944, 188.967, 38.142, -110.66, -235]
  MoveL 2439 to (19.12, -52.33, -277.46) mm, rotated rx -9.61 ry -16.54 rz 125.97 deg; joints [-16.192, -57.955, 111.848, 189.016, 38.011, -110.708, -235]
  MoveL 2440 to (20.99, -51.46, -277.4) mm, rotated rx -9.61 ry -16.54 rz 125.97 deg; joints [-16.181, -57.995, 111.745, 189.062, 37.87, -110.755, -235]
  MoveL 2441 to (22.95, -50.54, -277.33) mm, rotated rx -9.61 ry -16.54 rz 125.97 deg; joints [-16.169, -58.037, 111.637, 189.111, 37.724, -110.805, -235]
  MoveL 2442 to (25.08, -49.55, -277.18) mm, rotated rx -9.61 ry -16.54 rz 125.97 deg; joints [-16.153, -58.083, 111.52, 189.169, 37.564, -110.863, -235]
  MoveL 2443 to (26.78, -48.75, -277.07) mm, rotated rx -9.61 ry -16.54 rz 125.97 deg; joints [-16.141, -58.12, 111.427, 189.216, 37.437, -110.909, -235]
  MoveL 2444 to (28.94, -47.74, -276.85) mm, rotated rx -9.61 ry -16.54 rz 125.97 deg; joints [-16.122, -58.166, 111.309, 189.28, 37.277, -110.97, -235]
  MoveL 2445 to (30.64, -46.94, -276.74) mm, rotated rx -9.61 ry -16.54 rz 125.97 deg; joints [-16.11, -58.203, 111.216, 189.327, 37.15, -111.017, -235]
  MoveL 2446 to (32.57, -46.02, -276.57) mm, rotated rx -9.61 ry -16.54 rz 125.97 deg; joints [-16.094, -58.244, 111.11, 189.383, 37.007, -111.072, -235]
  MoveL 2447 to (34.73, -45, -276.52) mm, rotated rx -9.61 ry -16.54 rz 125.97 deg; joints [-16.082, -58.288, 110.989, 189.438, 36.844, -111.129, -235]
  MoveL 2448 to (36.43, -44.2, -276.41) mm, rotated rx -9.61 ry -16.54 rz 125.97 deg; joints [-16.07, -58.324, 110.895, 189.486, 36.718, -111.177, -235]
  MoveL 2449 to (38.35, -43.28, -276.25) mm, rotated rx -9.61 ry -16.54 rz 125.97 deg; joints [-16.055, -58.364, 110.788, 189.543, 36.574, -111.233, -235]
  MoveL 2450 to (40.51, -42.25, -276.2) mm, rotated rx -9.61 ry -16.54 rz 125.97 deg; joints [-16.043, -58.408, 110.666, 189.599, 36.412, -111.291, -235]
  MoveL 2451 to (42.21, -41.44, -276.09) mm, rotated rx -9.61 ry -16.54 rz 125.97 deg; joints [-16.031, -58.443, 110.572, 189.648, 36.286, -111.34, -235]
  MoveL 2452 to (44.21, -40.48, -275.98) mm, rotated rx -9.61 ry -16.54 rz 125.97 deg; joints [-16.018, -58.483, 110.459, 189.705, 36.136, -111.397, -235]
  MoveL 2453 to (46.22, -39.52, -275.92) mm, rotated rx -9.61 ry -16.54 rz 125.97 deg; joints [-16.006, -58.523, 110.345, 189.76, 35.986, -111.453, -235]
  MoveL 2454 to (47.9, -38.68, -275.74) mm, rotated rx -9.61 ry -16.54 rz 125.97 deg; joints [-15.991, -58.56, 110.253, 189.814, 35.86, -111.506, -235]
  MoveL 2455 to (49.44, -37.89, -275.48) mm, rotated rx -9.61 ry -16.54 rz 125.97 deg; joints [-15.975, -58.596, 110.171, 189.869, 35.746, -111.558, -235]
  MoveL 2456 to (50.87, -37.11, -275.13) mm, rotated rx -9.61 ry -16.54 rz 125.97 deg; joints [-15.955, -58.632, 110.098, 189.928, 35.64, -111.611, -235]
  MoveL 2457 to (49.38, -37.35, -274.44) mm, rotated rx -9.61 ry -16.54 rz 125.97 deg; joints [-15.936, -58.642, 110.215, 189.932, 35.748, -111.599, -235]
  MoveL 2458 to (49.6, -37.29, -274.44) mm, rotated rx -9.61 ry -16.54 rz 125.97 deg; joints [-15.935, -58.644, 110.201, 189.938, 35.733, -111.605, -235]
  MoveL 2459 to (49.9, -37.25, -274.42) mm, rotated rx -9.61 ry -16.54 rz 125.97 deg; joints [-15.932, -58.642, 110.179, 189.947, 35.713, -111.613, -235]
  MoveL 2460 to (50.35, -37.27, -274.39) mm, rotated rx -9.61 ry -16.54 rz 125.97 deg; joints [-15.928, -58.636, 110.144, 189.961, 35.685, -111.626, -235]
  MoveL 2461 to (50.89, -37.31, -274.35) mm, rotated rx -9.61 ry -16.54 rz 125.97 deg; joints [-15.923, -58.627, 110.102, 189.977, 35.653, -111.642, -235]
  MoveL 2462 to (51.5, -37.37, -274.31) mm, rotated rx -9.61 ry -16.54 rz 125.97 deg; joints [-15.917, -58.615, 110.053, 189.996, 35.617, -111.659, -235]
  MoveL 2463 to (54.09, -37.76, -274.31) mm, rotated rx -9.61 ry -16.54 rz 125.97 deg; joints [-15.898, -58.555, 109.837, 190.065, 35.465, -111.726, -235]
  MoveL 2464 to (54.7, -37.84, -274.28) mm, rotated rx -9.61 ry -16.54 rz 125.97 deg; joints [-15.892, -58.543, 109.788, 190.084, 35.43, -111.743, -235]
  MoveL 2465 to (55.38, -37.91, -274.22) mm, rotated rx -9.61 ry -16.54 rz 125.97 deg; joints [-15.885, -58.529, 109.733, 190.105, 35.39, -111.763, -235]
  MoveL 2466 to (56, -37.99, -274.19) mm, rotated rx -9.61 ry -16.54 rz 125.97 deg; joints [-15.88, -58.516, 109.682, 190.124, 35.353, -111.781, -235]
  MoveL 2467 to (56.52, -38.06, -274.19) mm, rotated rx -9.61 ry -16.54 rz 125.97 deg; joints [-15.876, -58.504, 109.639, 190.138, 35.323, -111.794, -235]
  MoveL 2468 to (57, -38.14, -274.18) mm, rotated rx -9.61 ry -16.54 rz 125.97 deg; joints [-15.872, -58.493, 109.598, 190.152, 35.294, -111.807, -235]
  MoveL 2469 to (57.52, -38.22, -274.18) mm, rotated rx -9.61 ry -16.54 rz 125.97 deg; joints [-15.868, -58.481, 109.555, 190.166, 35.264, -111.821, -235]
  MoveL 2470 to (58.03, -38.29, -274.18) mm, rotated rx -9.61 ry -16.54 rz 125.97 deg; joints [-15.864, -58.469, 109.512, 190.18, 35.234, -111.834, -235]
  MoveL 2471 to (58.51, -38.35, -274.15) mm, rotated rx -9.61 ry -16.54 rz 125.97 deg; joints [-15.86, -58.459, 109.473, 190.194, 35.206, -111.848, -235]
  MoveL 2472 to (58.97, -38.4, -274.1) mm, rotated rx -9.61 ry -16.54 rz 125.97 deg; joints [-15.855, -58.45, 109.436, 190.21, 35.179, -111.862, -235]
  MoveL 2473 to (59.46, -38.47, -274.09) mm, rotated rx -9.61 ry -16.54 rz 125.97 deg; joints [-15.851, -58.439, 109.395, 190.224, 35.15, -111.876, -235]
  MoveL 2474 to (59.99, -38.55, -274.08) mm, rotated rx -9.61 ry -16.54 rz 125.97 deg; joints [-15.847, -58.427, 109.351, 190.239, 35.119, -111.89, -235]
  MoveL 2475 to (61.03, -38.7, -274.08) mm, rotated rx -9.61 ry -16.54 rz 125.97 deg; joints [-15.839, -58.403, 109.264, 190.267, 35.059, -111.917, -235]
  Set speed (1000.0 mm/s)
  MoveL 2476 to (80.62, -47.84, -274.08) mm, rotated rx -9.61 ry -16.54 rz 125.97 deg; joints [-15.673, -57.523, 107.356, 190.82, 34.066, -112.433, -235]
  Print: /'Flow1'
  Set speed (1000.0 mm/s)
  MoveL 2477 to (40.38, 104.96, -81.82) mm, rotated rx 105.8 ry 33.04 rz -145.95 deg; joints [-3.332, -28.971, 98.058, 147.608, 81.185, 20.391, -295]
  Set speed (1000.0 mm/s)
  MoveL 2478 to (3.62, 79.22, -81.82) mm, rotated rx 105.8 ry 33.04 rz -145.95 deg; joints [-3.3, -29.88, 101.913, 147.848, 83.67, 18.796, -295]
  Set speed (100.0 mm/s)
  MoveL 2479 to (-55.98, 37.48, -81.82) mm, rotated rx 105.8 ry 33.04 rz -145.95 deg; joints [-3.244, -31.04, 107.839, 148.094, 87.703, 16.249, -295]
  MoveL 2480 to (-56.51, 37.51, -81.82) mm, rotated rx 105.8 ry 33.04 rz -145.95 deg; joints [-3.243, -31.067, 107.885, 148.095, 87.72, 16.238, -295]
  MoveL 2481 to (-57.15, 37.49, -81.72) mm, rotated rx 105.8 ry 33.04 rz -145.95 deg; joints [-3.239, -31.098, 107.943, 148.1, 87.743, 16.223, -295]
  MoveL 2482 to (-57.74, 37.49, -81.67) mm, rotated rx 105.8 ry 33.04 rz -145.95 deg; joints [-3.236, -31.127, 107.996, 148.104, 87.763, 16.21, -295]
  MoveL 2483 to (-58.31, 37.51, -81.64) mm, rotated rx 105.8 ry 33.04 rz -145.95 deg; joints [-3.234, -31.155, 108.047, 148.106, 87.781, 16.198, -295]
  MoveL 2484 to (-61.97, 37.71, -81.64) mm, rotated rx 105.8 ry 33.04 rz -145.95 deg; joints [-3.231, -31.344, 108.373, 148.112, 87.897, 16.125, -295]
  MoveL 2485 to (-63.41, 37.85, -81.73) mm, rotated rx 105.8 ry 33.04 rz -145.95 deg; joints [-3.233, -31.422, 108.501, 148.111, 87.941, 16.098, -295]
  MoveL 2486 to (-64.57, 38.09, -82) mm, rotated rx 105.8 ry 33.04 rz -145.95 deg; joints [-3.242, -31.491, 108.603, 148.102, 87.97, 16.082, -295]
  MoveL 2487 to (-65.45, 38.45, -82.44) mm, rotated rx 105.8 ry 33.04 rz -145.95 deg; joints [-3.26, -31.551, 108.68, 148.085, 87.986, 16.077, -295]
  MoveL 2488 to (-65.79, 38.66, -82.73) mm, rotated rx 105.8 ry 33.04 rz -145.95 deg; joints [-3.271, -31.578, 108.708, 148.074, 87.988, 16.079, -295]
  MoveL 2489 to (-66.05, 38.9, -83.06) mm, rotated rx 105.8 ry 33.04 rz -145.95 deg; joints [-3.285, -31.603, 108.73, 148.061, 87.987, 16.083, -295]
  MoveL 2490 to (-66.37, 39.46, -83.86) mm, rotated rx 105.8 ry 33.04 rz -145.95 deg; joints [-3.317, -31.646, 108.755, 148.029, 87.975, 16.098, -295]
  MoveL 2491 to (-66.4, 40.13, -84.84) mm, rotated rx 105.8 ry 33.04 rz -145.95 deg; joints [-3.357, -31.68, 108.753, 147.989, 87.95, 16.125, -295]
  MoveL 2492 to (-65.62, 41.79, -87.32) mm, rotated rx 105.8 ry 33.04 rz -145.95 deg; joints [-3.459, -31.723, 108.673, 147.886, 87.857, 16.21, -295]
  MoveL 2493 to (-64.05, 43.35, -89.81) mm, rotated rx 105.8 ry 33.04 rz -145.95 deg; joints [-3.562, -31.723, 108.522, 147.782, 87.743, 16.31, -295]
  MoveL 2494 to (-62.03, 44.32, -91.58) mm, rotated rx 105.8 ry 33.04 rz -145.95 deg; joints [-3.636, -31.671, 108.335, 147.707, 87.638, 16.396, -295]
  MoveL 2495 to (-60.86, 44.58, -92.2) mm, rotated rx 105.8 ry 33.04 rz -145.95 deg; joints [-3.662, -31.626, 108.229, 147.68, 87.589, 16.434, -295]
  MoveL 2496 to (-59.57, 44.68, -92.65) mm, rotated rx 105.8 ry 33.04 rz -145.95 deg; joints [-3.681, -31.568, 108.113, 147.66, 87.543, 16.469, -295]
  MoveL 2497 to (-56.67, 44.45, -93) mm, rotated rx 105.8 ry 33.04 rz -145.95 deg; joints [-3.698, -31.413, 107.855, 147.641, 87.457, 16.528, -295]
  MoveL 2498 to (-53.56, 43.92, -93.01) mm, rotated rx 105.8 ry 33.04 rz -145.95 deg; joints [-3.7, -31.235, 107.581, 147.636, 87.377, 16.58, -295]
  MoveL 2499 to (-53.08, 43.85, -93.03) mm, rotated rx 105.8 ry 33.04 rz -145.95 deg; joints [-3.701, -31.208, 107.538, 147.635, 87.363, 16.588, -295]
  MoveL 2500 to (-52.62, 43.8, -93.07) mm, rotated rx 105.8 ry 33.04 rz -145.95 deg; joints [-3.703, -31.183, 107.498, 147.632, 87.351, 16.597, -295]
  MoveL 2501 to (-52.21, 43.77, -93.13) mm, rotated rx 105.8 ry 33.04 rz -145.95 deg; joints [-3.706, -31.161, 107.461, 147.629, 87.338, 16.606, -295]
  MoveL 2502 to (-51.76, 43.73, -93.18) mm, rotated rx 105.8 ry 33.04 rz -145.95 deg; joints [-3.708, -31.137, 107.421, 147.627, 87.325, 16.614, -295]
  MoveL 2503 to (-51.22, 43.65, -93.2) mm, rotated rx 105.8 ry 33.04 rz -145.95 deg; joints [-3.71, -31.107, 107.373, 147.625, 87.311, 16.624, -295]
  MoveL 2504 to (-50.58, 43.56, -93.24) mm, rotated rx 105.8 ry 33.04 rz -145.95 deg; joints [-3.712, -31.071, 107.316, 147.622, 87.293, 16.636, -295]
  MoveL 2505 to (-50.02, 43.5, -93.3) mm, rotated rx 105.8 ry 33.04 rz -145.95 deg; joints [-3.715, -31.041, 107.267, 147.619, 87.277, 16.647, -295]
  MoveL 2506 to (-49.58, 43.47, -93.37) mm, rotated rx 105.8 ry 33.04 rz -145.95 deg; joints [-3.718, -31.017, 107.227, 147.615, 87.264, 16.656, -295]
  MoveL 2507 to (-49.14, 43.43, -93.42) mm, rotated rx 105.8 ry 33.04 rz -145.95 deg; joints [-3.72, -30.994, 107.188, 147.613, 87.251, 16.665, -295]
  MoveL 2508 to (-48.67, 43.36, -93.45) mm, rotated rx 105.8 ry 33.04 rz -145.95 deg; joints [-3.721, -30.967, 107.146, 147.611, 87.238, 16.673, -295]
  MoveL 2509 to (-48.15, 43.27, -93.45) mm, rotated rx 105.8 ry 33.04 rz -145.95 deg; joints [-3.722, -30.937, 107.1, 147.61, 87.225, 16.682, -295]
  MoveL 2510 to (-47.62, 43.18, -93.45) mm, rotated rx 105.8 ry 33.04 rz -145.95 deg; joints [-3.722, -30.907, 107.053, 147.61, 87.211, 16.691, -295]
  MoveL 2511 to (-47.05, 43.1, -93.46) mm, rotated rx 105.8 ry 33.04 rz -145.95 deg; joints [-3.723, -30.875, 107.003, 147.608, 87.195, 16.701, -295]
  MoveL 2512 to (-46.4, 43.02, -93.49) mm, rotated rx 105.8 ry 33.04 rz -145.95 deg; joints [-3.725, -30.839, 106.944, 147.606, 87.176, 16.714, -295]
  MoveL 2513 to (-45.81, 42.98, -93.56) mm, rotated rx 105.8 ry 33.04 rz -145.95 deg; joints [-3.728, -30.808, 106.891, 147.602, 87.158, 16.726, -295]
  MoveL 2514 to (-45.35, 42.98, -93.66) mm, rotated rx 105.8 ry 33.04 rz -145.95 deg; joints [-3.732, -30.785, 106.85, 147.597, 87.143, 16.737, -295]
  MoveL 2515 to (-45.35, 42.97, -93.9) mm, rotated rx 105.8 ry 33.04 rz -145.95 deg; joints [-3.742, -30.785, 106.851, 147.588, 87.145, 16.738, -295]
  MoveL 2516 to (-45.75, 42.91, -94.25) mm, rotated rx 105.8 ry 33.04 rz -145.95 deg; joints [-3.756, -30.802, 106.887, 147.575, 87.163, 16.731, -295]
  MoveL 2517 to (-46.36, 43.5, -95.22) mm, rotated rx 105.8 ry 33.04 rz -145.95 deg; joints [-3.795, -30.861, 106.938, 147.537, 87.162, 16.743, -295]
  MoveL 2518 to (-44.41, 44.37, -95.22) mm, rotated rx 105.8 ry 33.04 rz -145.95 deg; joints [-3.796, -30.804, 106.753, 147.532, 87.054, 16.812, -295]
  MoveL 2519 to (-42.33, 45.34, -95.35) mm, rotated rx 105.8 ry 33.04 rz -145.95 deg; joints [-3.802, -30.746, 106.556, 147.522, 86.937, 16.888, -295]
  MoveL 2520 to (-40.35, 46.24, -95.4) mm, rotated rx 105.8 ry 33.04 rz -145.95 deg; joints [-3.806, -30.688, 106.367, 147.515, 86.827, 16.959, -295]
  MoveL 2521 to (-38.42, 47.13, -95.53) mm, rotated rx 105.8 ry 33.04 rz -145.95 deg; joints [-3.812, -30.633, 106.183, 147.505, 86.719, 17.03, -295]
  MoveL 2522 to (-36.47, 48.02, -95.69) mm, rotated rx 105.8 ry 33.04 rz -145.95 deg; joints [-3.819, -30.577, 105.997, 147.494, 86.611, 17.101, -295]
  MoveL 2523 to (-34.54, 48.9, -95.81) mm, rotated rx 105.8 ry 33.04 rz -145.95 deg; joints [-3.825, -30.52, 105.812, 147.483, 86.503, 17.172, -295]
  MoveL 2524 to (-32.59, 49.8, -96.02) mm, rotated rx 105.8 ry 33.04 rz -145.95 deg; joints [-3.834, -30.463, 105.625, 147.47, 86.395, 17.243, -295]
  MoveL 2525 to (-30.66, 50.68, -96.14) mm, rotated rx 105.8 ry 33.04 rz -145.95 deg; joints [-3.84, -30.406, 105.44, 147.46, 86.288, 17.314, -295]
  MoveL 2526 to (-28.7, 51.56, -96.19) mm, rotated rx 105.8 ry 33.04 rz -145.95 deg; joints [-3.843, -30.347, 105.251, 147.452, 86.179, 17.384, -295]
  MoveL 2527 to (-26.73, 52.44, -96.34) mm, rotated rx 105.8 ry 33.04 rz -145.95 deg; joints [-3.85, -30.288, 105.062, 147.441, 86.071, 17.456, -295]
  MoveL 2528 to (-24.7, 53.36, -96.52) mm, rotated rx 105.8 ry 33.04 rz -145.95 deg; joints [-3.858, -30.227, 104.866, 147.428, 85.958, 17.53, -295]
  MoveL 2529 to (-22.67, 54.26, -96.7) mm, rotated rx 105.8 ry 33.04 rz -145.95 deg; joints [-3.867, -30.164, 104.67, 147.415, 85.847, 17.605, -295]
  MoveL 2530 to (-20.95, 55.02, -96.94) mm, rotated rx 105.8 ry 33.04 rz -145.95 deg; joints [-3.877, -30.112, 104.505, 147.4, 85.753, 17.668, -295]
  MoveL 2531 to (-18.52, 56.11, -97.05) mm, rotated rx 105.8 ry 33.04 rz -145.95 deg; joints [-3.882, -30.036, 104.268, 147.388, 85.618, 17.756, -295]
  Set speed (1000.0 mm/s)
  MoveL 2532 to (18.59, 82.09, -97.05) mm, rotated rx 105.8 ry 33.04 rz -145.95 deg; joints [-3.898, -29.23, 100.489, 147.214, 83.119, 19.374, -295]
  Set speed (1000.0 mm/s)
  MoveL 2533 to (21.88, 77.39, -108.93) mm, rotated rx 105.8 ry 33.04 rz -145.95 deg; joints [-4.357, -28.869, 100.245, 146.773, 83.297, 19.434, -295]
  Set speed (100.0 mm/s)
  MoveL 2534 to (-1.62, 60.94, -108.93) mm, rotated rx 105.8 ry 33.04 rz -145.95 deg; joints [-4.356, -29.394, 102.657, 146.881, 84.876, 18.395, -295]
  MoveL 2535 to (-3.27, 60.46, -108.68) mm, rotated rx 105.8 ry 33.04 rz -145.95 deg; joints [-4.346, -29.458, 102.816, 146.895, 84.954, 18.341, -295]
  MoveL 2536 to (-5.2, 59.86, -108.62) mm, rotated rx 105.8 ry 33.04 rz -145.95 deg; joints [-4.343, -29.531, 103.003, 146.904, 85.049, 18.278, -295]
  MoveL 2537 to (-7.16, 59.26, -108.47) mm, rotated rx 105.8 ry 33.04 rz -145.95 deg; joints [-4.337, -29.605, 103.192, 146.915, 85.145, 18.213, -295]
  MoveL 2538 to (-9.52, 58.55, -108.34) mm, rotated rx 105.8 ry 33.04 rz -145.95 deg; joints [-4.331, -29.695, 103.419, 146.927, 85.259, 18.137, -295]
  MoveL 2539 to (-11.56, 57.92, -108.34) mm, rotated rx 105.8 ry 33.04 rz -145.95 deg; joints [-4.331, -29.771, 103.615, 146.932, 85.359, 18.071, -295]
  MoveL 2540 to (-13.81, 57.21, -108.18) mm, rotated rx 105.8 ry 33.04 rz -145.95 deg; joints [-4.324, -29.855, 103.832, 146.945, 85.469, 17.997, -295]
  MoveL 2541 to (-15.71, 56.63, -108) mm, rotated rx 105.8 ry 33.04 rz -145.95 deg; joints [-4.316, -29.926, 104.014, 146.957, 85.561, 17.934, -295]
  MoveL 2542 to (-17.67, 56.03, -107.9) mm, rotated rx 105.8 ry 33.04 rz -145.95 deg; joints [-4.312, -29.999, 104.202, 146.966, 85.657, 17.871, -295]
  MoveL 2543 to (-19.71, 55.39, -107.69) mm, rotated rx 105.8 ry 33.04 rz -145.95 deg; joints [-4.303, -30.074, 104.396, 146.98, 85.756, 17.803, -295]
  MoveL 2544 to (-21.72, 54.76, -107.53) mm, rotated rx 105.8 ry 33.04 rz -145.95 deg; joints [-4.296, -30.148, 104.588, 146.991, 85.854, 17.737, -295]
  MoveL 2545 to (-23.74, 54.12, -107.42) mm, rotated rx 105.8 ry 33.04 rz -145.95 deg; joints [-4.292, -30.221, 104.781, 147, 85.953, 17.671, -295]
  MoveL 2546 to (-25.78, 53.47, -107.25) mm, rotated rx 105.8 ry 33.04 rz -145.95 deg; joints [-4.285, -30.295, 104.975, 147.012, 86.053, 17.604, -295]
  MoveL 2547 to (-27.8, 52.82, -107.11) mm, rotated rx 105.8 ry 33.04 rz -145.95 deg; joints [-4.278, -30.368, 105.167, 147.022, 86.152, 17.537, -295]
  MoveL 2548 to (-29.88, 52.17, -107.04) mm, rotated rx 105.8 ry 33.04 rz -145.95 deg; joints [-4.275, -30.444, 105.364, 147.03, 86.254, 17.47, -295]
  MoveL 2549 to (-31.91, 51.5, -106.83) mm, rotated rx 105.8 ry 33.04 rz -145.95 deg; joints [-4.267, -30.515, 105.556, 147.042, 86.354, 17.403, -295]
  MoveL 2550 to (-33.92, 50.85, -106.71) mm, rotated rx 105.8 ry 33.04 rz -145.95 deg; joints [-4.261, -30.587, 105.747, 147.052, 86.453, 17.337, -295]
  MoveL 2551 to (-35.98, 50.18, -106.59) mm, rotated rx 105.8 ry 33.04 rz -145.95 deg; joints [-4.256, -30.66, 105.942, 147.061, 86.554, 17.269, -295]
  MoveL 2552 to (-37.62, 49.51, -106.38) mm, rotated rx 105.8 ry 33.04 rz -145.95 deg; joints [-4.247, -30.712, 106.098, 147.073, 86.64, 17.211, -295]
  MoveL 2553 to (-38.93, 48.83, -106.03) mm, rotated rx 105.8 ry 33.04 rz -145.95 deg; joints [-4.233, -30.746, 106.223, 147.09, 86.715, 17.158, -295]
  MoveL 2554 to (-39.9, 48.11, -105.5) mm, rotated rx 105.8 ry 33.04 rz -145.95 deg; joints [-4.211, -30.761, 106.318, 147.113, 86.779, 17.11, -295]
  MoveL 2555 to (-38.36, 48.11, -104.64) mm, rotated rx 105.8 ry 33.04 rz -145.95 deg; joints [-4.177, -30.683, 106.178, 147.145, 86.722, 17.137, -295]
  MoveL 2556 to (-39.16, 48.04, -104.64) mm, rotated rx 105.8 ry 33.04 rz -145.95 deg; joints [-4.177, -30.72, 106.251, 147.146, 86.753, 17.117, -295]
  MoveL 2557 to (-39.86, 48.04, -104.64) mm, rotated rx 105.8 ry 33.04 rz -145.95 deg; joints [-4.177, -30.755, 106.315, 147.147, 86.777, 17.101, -295]
  MoveL 2558 to (-40.49, 48.14, -104.64) mm, rotated rx 105.8 ry 33.04 rz -145.95 deg; joints [-4.176, -30.791, 106.371, 147.148, 86.794, 17.09, -295]
  MoveL 2559 to (-41.14, 48.28, -104.62) mm, rotated rx 105.8 ry 33.04 rz -145.95 deg; joints [-4.175, -30.83, 106.429, 147.15, 86.809, 17.08, -295]
  MoveL 2560 to (-41.89, 48.47, -104.58) mm, rotated rx 105.8 ry 33.04 rz -145.95 deg; joints [-4.174, -30.876, 106.494, 147.152, 86.826, 17.069, -295]
  MoveL 2561 to (-43.89, 49.07, -104.58) mm, rotated rx 105.8 ry 33.04 rz -145.95 deg; joints [-4.173, -31.004, 106.671, 147.155, 86.866, 17.042, -295]
  MoveL 2562 to (-44.32, 49.18, -104.56) mm, rotated rx 105.8 ry 33.04 rz -145.95 deg; joints [-4.172, -31.03, 106.708, 147.156, 86.875, 17.036, -295]
  MoveL 2563 to (-45.33, 49.48, -104.56) mm, rotated rx 105.8 ry 33.04 rz -145.95 deg; joints [-4.171, -31.094, 106.796, 147.157, 86.895, 17.023, -295]
  MoveL 2564 to (-45.81, 49.62, -104.56) mm, rotated rx 105.8 ry 33.04 rz -145.95 deg; joints [-4.171, -31.125, 106.839, 147.158, 86.905, 17.016, -295]
  MoveL 2565 to (-46.29, 49.75, -104.54) mm, rotated rx 105.8 ry 33.04 rz -145.95 deg; joints [-4.17, -31.154, 106.88, 147.159, 86.915, 17.01, -295]
  MoveL 2566 to (-46.75, 49.87, -104.51) mm, rotated rx 105.8 ry 33.04 rz -145.95 deg; joints [-4.168, -31.183, 106.921, 147.161, 86.925, 17.003, -295]
  MoveL 2567 to (-47.18, 49.95, -104.45) mm, rotated rx 105.8 ry 33.04 rz -145.95 deg; joints [-4.166, -31.208, 106.959, 147.164, 86.936, 16.995, -295]
  MoveL 2568 to (-47.64, 50.06, -104.41) mm, rotated rx 105.8 ry 33.04 rz -145.95 deg; joints [-4.164, -31.236, 106.999, 147.166, 86.946, 16.988, -295]
  MoveL 2569 to (-48.11, 50.19, -104.39) mm, rotated rx 105.8 ry 33.04 rz -145.95 deg; joints [-4.163, -31.266, 107.041, 147.167, 86.956, 16.982, -295]
  MoveL 2570 to (-48.6, 50.33, -104.39) mm, rotated rx 105.8 ry 33.04 rz -145.95 deg; joints [-4.162, -31.297, 107.084, 147.168, 86.966, 16.975, -295]
  MoveL 2571 to (-49.08, 50.46, -104.37) mm, rotated rx 105.8 ry 33.04 rz -145.95 deg; joints [-4.161, -31.326, 107.125, 147.17, 86.976, 16.968, -295]
  MoveL 2572 to (-49.55, 50.57, -104.33) mm, rotated rx 105.8 ry 33.04 rz -145.95 deg; joints [-4.16, -31.355, 107.166, 147.171, 86.986, 16.961, -295]
  MoveL 2573 to (-49.97, 50.65, -104.28) mm, rotated rx 105.8 ry 33.04 rz -145.95 deg; joints [-4.157, -31.379, 107.204, 147.174, 86.996, 16.954, -295]
  MoveL 2574 to (-50.42, 50.74, -104.22) mm, rotated rx 105.8 ry 33.04 rz -145.95 deg; joints [-4.155, -31.406, 107.243, 147.177, 87.007, 16.946, -295]
  MoveL 2575 to (-51.82, 51.08, -104.14) mm, rotated rx 105.8 ry 33.04 rz -145.95 deg; joints [-4.151, -31.491, 107.366, 147.182, 87.038, 16.925, -295]
  MoveL 2576 to (-52.92, 51.5, -104.27) mm, rotated rx 105.8 ry 33.04 rz -145.95 deg; joints [-4.155, -31.566, 107.46, 147.178, 87.055, 16.915, -295]
  MoveL 2577 to (-53.72, 52, -104.6) mm, rotated rx 105.8 ry 33.04 rz -145.95 deg; joints [-4.169, -31.629, 107.528, 147.165, 87.06, 16.916, -295]
  MoveL 2578 to (-54, 52.28, -104.85) mm, rotated rx 105.8 ry 33.04 rz -145.95 deg; joints [-4.178, -31.656, 107.551, 147.155, 87.058, 16.92, -295]
  MoveL 2579 to (-54.22, 52.58, -105.15) mm, rotated rx 105.8 ry 33.04 rz -145.95 deg; joints [-4.19, -31.681, 107.567, 147.143, 87.053, 16.927, -295]
  MoveL 2580 to (-54.42, 53.24, -105.91) mm, rotated rx 105.8 ry 33.04 rz -145.95 deg; joints [-4.221, -31.722, 107.579, 147.113, 87.032, 16.949, -295]
  MoveL 2581 to (-54.33, 53.97, -106.88) mm, rotated rx 105.8 ry 33.04 rz -145.95 deg; joints [-4.26, -31.752, 107.564, 147.073, 87, 16.981, -295]
  MoveL 2582 to (-53.25, 55.66, -109.44) mm, rotated rx 105.8 ry 33.04 rz -145.95 deg; joints [-4.363, -31.778, 107.45, 146.968, 86.896, 17.079, -295]
  MoveL 2583 to (-51.41, 57.12, -112.05) mm, rotated rx 105.8 ry 33.04 rz -145.95 deg; joints [-4.469, -31.755, 107.27, 146.86, 86.779, 17.187, -295]
  MoveL 2584 to (-50.38, 57.56, -113.08) mm, rotated rx 105.8 ry 33.04 rz -145.95 deg; joints [-4.511, -31.724, 107.173, 146.817, 86.729, 17.232, -295]
  MoveL 2585 to (-49.27, 57.81, -113.92) mm, rotated rx 105.8 ry 33.04 rz -145.95 deg; joints [-4.544, -31.68, 107.071, 146.782, 86.685, 17.271, -295]
  MoveL 2586 to (-48.09, 57.85, -114.57) mm, rotated rx 105.8 ry 33.04 rz -145.95 deg; joints [-4.571, -31.623, 106.963, 146.754, 86.646, 17.305, -295]
  MoveL 2587 to (-46.82, 57.71, -115.04) mm, rotated rx 105.8 ry 33.04 rz -145.95 deg; joints [-4.59, -31.553, 106.851, 146.734, 86.613, 17.332, -295]
  MoveL 2588 to (-45.48, 57.37, -115.32) mm, rotated rx 105.8 ry 33.04 rz -145.95 deg; joints [-4.602, -31.471, 106.733, 146.722, 86.586, 17.354, -295]
  MoveL 2589 to (-44.07, 56.83, -115.41) mm, rotated rx 105.8 ry 33.04 rz -145.95 deg; joints [-4.606, -31.375, 106.611, 146.717, 86.564, 17.369, -295]
  MoveL 2590 to (-41.17, 55.57, -115.41) mm, rotated rx 105.8 ry 33.04 rz -145.95 deg; joints [-4.607, -31.172, 106.361, 146.714, 86.525, 17.395, -295]
  MoveL 2591 to (-40.66, 55.36, -115.43) mm, rotated rx 105.8 ry 33.04 rz -145.95 deg; joints [-4.607, -31.137, 106.317, 146.713, 86.518, 17.4, -295]
  MoveL 2592 to (-40.08, 55.13, -115.46) mm, rotated rx 105.8 ry 33.04 rz -145.95 deg; joints [-4.609, -31.097, 106.267, 146.711, 86.509, 17.406, -295]
  MoveL 2593 to (-39.36, 54.89, -115.56) mm, rotated rx 105.8 ry 33.04 rz -145.95 deg; joints [-4.613, -31.05, 106.204, 146.707, 86.497, 17.416, -295]
  MoveL 2594 to (-38.78, 54.66, -115.59) mm, rotated rx 105.8 ry 33.04 rz -145.95 deg; joints [-4.615, -31.011, 106.154, 146.705, 86.488, 17.422, -295]
  MoveL 2595 to (-38.28, 54.45, -115.61) mm, rotated rx 105.8 ry 33.04 rz -145.95 deg; joints [-4.615, -30.976, 106.111, 146.704, 86.481, 17.427, -295]
  MoveL 2596 to (-37.81, 54.26, -115.62) mm, rotated rx 105.8 ry 33.04 rz -145.95 deg; joints [-4.616, -30.944, 106.07, 146.703, 86.474, 17.431, -295]
  MoveL 2597 to (-37.39, 54.08, -115.63) mm, rotated rx 105.8 ry 33.04 rz -145.95 deg; joints [-4.616, -30.914, 106.033, 146.702, 86.468, 17.436, -295]
  MoveL 2598 to (-35.5, 53.27, -115.64) mm, rotated rx 105.8 ry 33.04 rz -145.95 deg; joints [-4.617, -30.782, 105.87, 146.7, 86.442, 17.453, -295]
  MoveL 2599 to (-35.02, 53.09, -115.68) mm, rotated rx 105.8 ry 33.04 rz -145.95 deg; joints [-4.619, -30.75, 105.828, 146.698, 86.434, 17.459, -295]
  MoveL 2600 to (-34.57, 52.93, -115.73) mm, rotated rx 105.8 ry 33.04 rz -145.95 deg; joints [-4.621, -30.721, 105.789, 146.696, 86.426, 17.465, -295]
  MoveL 2601 to (-34.13, 52.8, -115.8) mm, rotated rx 105.8 ry 33.04 rz -145.95 deg; joints [-4.624, -30.692, 105.75, 146.693, 86.418, 17.471, -295]
  MoveL 2602 to (-33.66, 52.68, -115.86) mm, rotated rx 105.8 ry 33.04 rz -145.95 deg; joints [-4.627, -30.663, 105.708, 146.69, 86.408, 17.479, -295]
  MoveL 2603 to (-33.12, 52.56, -115.89) mm, rotated rx 105.8 ry 33.04 rz -145.95 deg; joints [-4.628, -30.631, 105.66, 146.688, 86.395, 17.487, -295]
  MoveL 2604 to (-32.45, 52.51, -115.9) mm, rotated rx 105.8 ry 33.04 rz -145.95 deg; joints [-4.628, -30.595, 105.599, 146.687, 86.374, 17.501, -295]
  MoveL 2605 to (-31.68, 52.52, -115.9) mm, rotated rx 105.8 ry 33.04 rz -145.95 deg; joints [-4.629, -30.556, 105.529, 146.685, 86.347, 17.519, -295]
  MoveL 2606 to (-33.4, 53.42, -117.46) mm, rotated rx 105.8 ry 33.04 rz -145.95 deg; joints [-4.69, -30.684, 105.677, 146.626, 86.373, 17.521, -295]
  MoveL 2607 to (-31.08, 53.87, -117.59) mm, rotated rx 105.8 ry 33.04 rz -145.95 deg; joints [-4.695, -30.588, 105.46, 146.616, 86.273, 17.589, -295]
  MoveL 2608 to (-28.88, 54.29, -117.7) mm, rotated rx 105.8 ry 33.04 rz -145.95 deg; joints [-4.7, -30.496, 105.255, 146.608, 86.179, 17.652, -295]
  MoveL 2609 to (-26.77, 54.71, -117.86) mm, rotated rx 105.8 ry 33.04 rz -145.95 deg; joints [-4.706, -30.408, 105.056, 146.598, 86.088, 17.715, -295]
  MoveL 2610 to (-24.67, 55.11, -117.97) mm, rotated rx 105.8 ry 33.04 rz -145.95 deg; joints [-4.71, -30.32, 104.86, 146.589, 85.998, 17.775, -295]
  MoveL 2611 to (-22.57, 55.51, -118.08) mm, rotated rx 105.8 ry 33.04 rz -145.95 deg; joints [-4.715, -30.231, 104.662, 146.581, 85.907, 17.836, -295]
  MoveL 2612 to (-20.48, 55.92, -118.3) mm, rotated rx 105.8 ry 33.04 rz -145.95 deg; joints [-4.723, -30.144, 104.465, 146.568, 85.817, 17.899, -295]
  MoveL 2613 to (-18.38, 56.33, -118.52) mm, rotated rx 105.8 ry 33.04 rz -145.95 deg; joints [-4.732, -30.055, 104.267, 146.555, 85.727, 17.961, -295]
  MoveL 2614 to (-16.28, 56.72, -118.64) mm, rotated rx 105.8 ry 33.04 rz -145.95 deg; joints [-4.736, -29.966, 104.069, 146.546, 85.637, 18.022, -295]
  MoveL 2615 to (-14.18, 57.1, -118.64) mm, rotated rx 105.8 ry 33.04 rz -145.95 deg; joints [-4.736, -29.876, 103.871, 146.542, 85.547, 18.082, -295]
  MoveL 2616 to (-12.08, 57.49, -118.75) mm, rotated rx 105.8 ry 33.04 rz -145.95 deg; joints [-4.741, -29.786, 103.672, 146.533, 85.457, 18.143, -295]
  MoveL 2617 to (-9.96, 57.88, -118.95) mm, rotated rx 105.8 ry 33.04 rz -145.95 deg; joints [-4.749, -29.694, 103.47, 146.52, 85.366, 18.206, -295]
  MoveL 2618 to (-7.97, 58.24, -119.13) mm, rotated rx 105.8 ry 33.04 rz -145.95 deg; joints [-4.756, -29.609, 103.282, 146.509, 85.281, 18.265, -295]
  MoveL 2619 to (-6.15, 58.58, -119.35) mm, rotated rx 105.8 ry 33.04 rz -145.95 deg; joints [-4.764, -29.53, 103.108, 146.496, 85.204, 18.319, -295]
  MoveL 2620 to (-4.22, 58.93, -119.44) mm, rotated rx 105.8 ry 33.04 rz -145.95 deg; joints [-4.767, -29.446, 102.924, 146.488, 85.12, 18.376, -295]
